C01791=1018.600,222.779,-127.632,168.817,51.228,159.725
C01792=1018.606,223.027,-127.658,168.821,51.221,159.724
C01793=1018.612,223.276,-127.684,168.825,51.214,159.724
C01794=1018.618,223.524,-127.710,168.829,51.207,159.723
C01795=1018.624,223.773,-127.736,168.833,51.201,159.722
C01796=1018.631,224.022,-127.763,168.836,51.194,159.721
C01797=1018.636,224.271,-127.789,168.841,51.188,159.721
C01798=1018.643,224.519,-127.815,168.846,51.181,159.720
C01799=1018.648,224.768,-127.841,168.849,51.174,159.719
C01800=1018.655,225.016,-127.867,168.854,51.168,159.719
C01801=1018.660,225.265,-127.893,168.857,51.161,159.718
C01802=1018.666,225.513,-127.919,168.862,51.155,159.717
C01803=1018.672,225.761,-127.945,168.865,51.148,159.716
C01804=1018.678,226.010,-127.971,168.870,51.141,159.716
C01805=1018.684,226.258,-127.997,168.873,51.135,159.715
C01806=1018.690,226.508,-128.024,168.877,51.128,159.714
C01807=1018.696,226.756,-128.050,168.881,51.122,159.714
C01808=1018.702,227.005,-128.077,168.886,51.115,159.713
C01809=1018.709,227.253,-128.103,168.889,51.109,159.712
C01810=1018.714,227.502,-128.129,168.894,51.102,159.712
C01811=1018.720,227.750,-128.156,168.897,51.096,159.711
C01812=1018.726,227.998,-128.182,168.902,51.090,159.710
C01813=1018.731,228.247,-128.209,168.906,51.083,159.710
C01814=1018.738,228.496,-128.236,168.910,51.077,159.709
C01815=1018.743,228.745,-128.262,168.914,51.071,159.709
C01816=1018.750,228.993,-128.288,168.918,51.064,159.708
C01817=1018.755,229.241,-128.314,168.922,51.058,159.707
C01818=1018.761,229.490,-128.341,168.927,51.051,159.706
C01819=1018.767,229.738,-128.368,168.930,51.045,159.706
C01820=1018.773,229.987,-128.395,168.935,51.039,159.705
C01821=1018.779,230.235,-128.421,168.939,51.033,159.705
C01822=1018.785,230.484,-128.448,168.942,51.026,159.704
C01823=1018.791,230.732,-128.475,168.947,51.020,159.703
C01824=1018.796,230.980,-128.501,168.951,51.014,159.703
C01825=1018.803,231.229,-128.528,168.955,51.007,159.702
C01826=1018.808,231.478,-128.554,168.959,51.001,159.701
C01827=1018.814,231.727,-128.581,168.964,50.995,159.701
C01828=1018.820,231.975,-128.608,168.967,50.989,159.700
C01829=1018.826,232.223,-128.635,168.971,50.983,159.699
C01830=1018.832,232.472,-128.662,168.976,50.976,159.699
C01831=1018.838,232.720,-128.689,168.979,50.970,159.698
C01832=1018.844,232.969,-128.715,168.984,50.964,159.698
C01833=1018.850,233.217,-128.742,168.988,50.958,159.697
C01834=1018.856,233.444,-128.766,168.992,50.952,159.697
C01835=1018.861,233.670,-128.790,168.996,50.947,159.696
C01836=1018.867,233.895,-128.815,169.000,50.941,159.695
C01837=1018.872,234.122,-128.839,169.003,50.936,159.695
C01838=1018.877,234.348,-128.864,169.007,50.930,159.694
C01839=1018.882,234.574,-128.888,169.011,50.924,159.694
C01840=1018.888,234.800,-128.913,169.015,50.919,159.693
C01841=1018.893,235.026,-128.937,169.019,50.913,159.693
C01842=1018.900,235.275,-128.964,169.022,50.907,159.692
C01843=1018.905,235.523,-128.991,169.027,50.901,159.692
C01844=1018.911,235.771,-129.018,169.031,50.895,159.691
C01845=1018.917,236.019,-129.045,169.034,50.889,159.690
C01846=1018.924,236.268,-129.072,169.040,50.883,159.690
C01847=1018.929,236.517,-129.098,169.043,50.877,159.689
C01848=1018.936,236.766,-129.125,169.047,50.871,159.688
C01849=1018.942,237.014,-129.153,169.052,50.864,159.688
C01850=1018.948,237.262,-129.179,169.056,50.859,159.687
C01851=1018.954,237.511,-129.206,169.060,50.852,159.687
C01852=1018.960,237.759,-129.234,169.064,50.846,159.686
C01853=1018.966,238.007,-129.260,169.068,50.840,159.686
C01854=1018.972,238.256,-129.287,169.073,50.834,159.685
C01855=1018.978,238.504,-129.314,169.077,50.828,159.684
C01856=1018.985,238.753,-129.342,169.080,50.822,159.684
C01857=1018.990,239.002,-129.369,169.085,50.817,159.683
C01858=1018.996,239.249,-129.396,169.089,50.810,159.683
C01859=1019.002,239.498,-129.423,169.093,50.805,159.682
C01860=1019.008,239.747,-129.450,169.098,50.799,159.682
C01861=1019.014,239.996,-129.478,169.102,50.793,159.681
C01862=1019.020,240.244,-129.505,169.106,50.787,159.681
C01863=1019.026,240.492,-129.532,169.111,50.781,159.680
C01864=1019.032,240.740,-129.561,169.114,50.775,159.680
C01865=1019.037,240.989,-129.587,169.119,50.770,159.679
C01866=1019.044,241.237,-129.615,169.123,50.764,159.678
C01867=1019.049,241.486,-129.642,169.127,50.758,159.678
C01868=1019.056,241.734,-129.670,169.131,50.752,159.677
C01869=1019.061,241.983,-129.697,169.135,50.747,159.677
C01870=1019.067,242.231,-129.725,169.140,50.741,159.676
C01871=1019.073,242.480,-129.752,169.144,50.735,159.676
C01872=1019.079,242.728,-129.780,169.148,50.730,159.675
C01873=1019.085,242.976,-129.807,169.153,50.723,159.675
C01874=1019.091,243.225,-129.834,169.157,50.718,159.674
C01875=1019.097,243.473,-129.862,169.161,50.712,159.674
C01876=1019.102,243.721,-129.890,169.165,50.707,159.673
C01877=1019.109,243.970,-129.918,169.170,50.701,159.673
C01878=1019.114,244.218,-129.946,169.174,50.695,159.672
C01879=1019.121,244.467,-129.973,169.178,50.690,159.672
C01880=1019.126,244.715,-130.001,169.182,50.684,159.671
C01881=1019.132,244.964,-130.029,169.187,50.679,159.671
C01882=1019.138,245.211,-130.057,169.191,50.673,159.670
C01883=1019.144,245.460,-130.085,169.195,50.667,159.670
C01884=1019.149,245.708,-130.113,169.199,50.662,159.669
C01885=1019.156,245.957,-130.140,169.203,50.657,159.669
C01886=1019.161,246.205,-130.168,169.208,50.651,159.669
C01887=1019.168,246.454,-130.196,169.213,50.645,159.668
C01888=1019.174,246.703,-130.224,169.217,50.640,159.668
C01889=1019.179,246.951,-130.252,169.221,50.635,159.667
C01890=1019.186,247.199,-130.280,169.226,50.628,159.667
C01891=1019.191,247.447,-130.308,169.230,50.623,159.666
C01892=1019.197,247.696,-130.336,169.234,50.618,159.666
C01893=1019.203,247.944,-130.363,169.238,50.612,159.665
C01894=1019.208,248.167,-130.389,169.242,50.608,159.665
C01895=1019.213,248.390,-130.413,169.245,50.602,159.664
C01896=1019.219,248.612,-130.438,169.250,50.598,159.664
C01897=1019.224,248.835,-130.464,169.253,50.593,159.663
C01898=1019.230,249.058,-130.489,169.258,50.588,159.663
C01899=1019.235,249.280,-130.514,169.262,50.583,159.663
C01900=1019.241,249.504,-130.539,169.265,50.578,159.662
C01901=1019.246,249.726,-130.564,169.269,50.573,159.662
C01902=1019.252,249.975,-130.592,169.273,50.568,159.661
C01903=1019.258,250.224,-130.620,169.278,50.562,159.661
C01904=1019.264,250.472,-130.648,169.282,50.557,159.660
C01905=1019.271,250.720,-130.677,169.287,50.551,159.660
C01906=1019.276,250.968,-130.705,169.291,50.546,159.660
C01907=1019.282,251.216,-130.733,169.295,50.541,159.659
C01908=1019.288,251.465,-130.761,169.300,50.536,159.659
C01909=1019.294,251.714,-130.789,169.305,50.530,159.659
C01910=1019.300,251.962,-130.817,169.309,50.525,159.658
C01911=1019.306,252.210,-130.845,169.313,50.519,159.658
C01912=1019.312,252.459,-130.873,169.317,50.514,159.657
C01913=1019.319,252.707,-130.902,169.321,50.509,159.657
C01914=1019.325,252.955,-130.930,169.326,50.503,159.656
C01915=1019.331,253.203,-130.958,169.331,50.498,159.656
C01916=1019.337,253.452,-130.986,169.335,50.493,159.656
C01917=1019.344,253.700,-131.014,169.339,50.488,159.655
C01918=1019.350,253.949,-131.043,169.343,50.482,159.655
C01919=1019.356,254.196,-131.070,169.348,50.477,159.654
C01920=1019.362,254.445,-131.098,169.352,50.471,159.654
C01921=1019.368,254.693,-131.128,169.357,50.466,159.653
C01922=1019.375,254.942,-131.155,169.361,50.461,159.653
C01923=1019.380,255.191,-131.184,169.366,50.455,159.653
C01924=1019.386,255.439,-131.212,169.370,50.450,159.652
C01925=1019.393,255.686,-131.240,169.375,50.445,159.652
C01926=1019.399,255.935,-131.268,169.379,50.440,159.651
C01927=1019.405,256.184,-131.297,169.383,50.435,159.651
C01928=1019.412,256.432,-131.325,169.388,50.429,159.650
C01929=1019.418,256.680,-131.353,169.393,50.424,159.650
C01930=1019.423,256.929,-131.381,169.397,50.419,159.650
C01931=1019.430,257.176,-131.410,169.401,50.414,159.649
C01932=1019.436,257.425,-131.438,169.406,50.409,159.649
C01933=1019.442,257.673,-131.467,169.411,50.403,159.649
C01934=1019.449,257.922,-131.495,169.415,50.398,159.648
C01935=1019.455,258.170,-131.524,169.419,50.393,159.648
C01936=1019.461,258.419,-131.552,169.423,50.388,159.647
C01937=1019.468,258.667,-131.580,169.429,50.383,159.647
C01938=1019.474,258.915,-131.609,169.433,50.378,159.647
C01939=1019.480,259.164,-131.637,169.437,50.372,159.646
C01940=1019.487,259.412,-131.666,169.442,50.368,159.646
C01941=1019.492,259.660,-131.694,169.446,50.362,159.645
C01942=1019.498,259.908,-131.723,169.451,50.357,159.645
C01943=1019.505,260.156,-131.752,169.456,50.352,159.645
C01944=1019.511,260.405,-131.780,169.460,50.347,159.645
C01945=1019.517,260.653,-131.809,169.464,50.342,159.644
C01946=1019.523,260.901,-131.838,169.469,50.337,159.644
C01947=1019.529,261.149,-131.867,169.473,50.333,159.644
C01948=1019.535,261.398,-131.896,169.477,50.327,159.643
C01949=1019.542,261.646,-131.925,169.482,50.323,159.643
C01950=1019.548,261.894,-131.954,169.487,50.318,159.643
C01951=1019.554,262.142,-131.983,169.492,50.313,159.642
C01952=1019.560,262.390,-132.012,169.496,50.308,159.642
C01953=1019.566,262.639,-132.040,169.501,50.303,159.642
C01954=1019.571,262.861,-132.066,169.504,50.299,159.641
C01955=1019.577,263.083,-132.092,169.509,50.294,159.641
C01956=1019.582,263.305,-132.118,169.513,50.290,159.641
C01957=1019.588,263.527,-132.144,169.517,50.286,159.641
C01958=1019.593,263.749,-132.170,169.521,50.281,159.640
C01959=1019.599,263.970,-132.196,169.525,50.277,159.640
C01960=1019.605,264.192,-132.222,169.529,50.272,159.639
C01961=1019.610,264.415,-132.248,169.534,50.268,159.639
C01962=1019.616,264.663,-132.277,169.538,50.263,159.639
C01963=1019.622,264.911,-132.306,169.542,50.259,159.639
C01964=1019.629,265.159,-132.335,169.547,50.254,159.638
C01965=1019.635,265.407,-132.364,169.551,50.249,159.638
C01966=1019.640,265.656,-132.394,169.556,50.245,159.638
C01967=1019.647,265.904,-132.423,169.560,50.240,159.638
C01968=1019.653,266.152,-132.452,169.566,50.235,159.637
C01969=1019.659,266.400,-132.481,169.570,50.230,159.637
C01970=1019.665,266.648,-132.510,169.575,50.226,159.637
C01971=1019.671,266.896,-132.540,169.579,50.221,159.637
C01972=1019.678,267.145,-132.570,169.584,50.216,159.636
C01973=1019.684,267.393,-132.599,169.589,50.212,159.636
C01974=1019.691,267.641,-132.628,169.593,50.207,159.636
C01975=1019.696,267.890,-132.657,169.598,50.202,159.635
C01976=1019.702,268.138,-132.686,169.602,50.198,159.635
C01977=1019.709,268.385,-132.716,169.607,50.193,159.635
C01978=1019.714,268.634,-132.746,169.612,50.188,159.635
C01979=1019.721,268.882,-132.775,169.617,50.183,159.634
C01980=1019.727,269.131,-132.804,169.621,50.179,159.634
C01981=1019.734,269.379,-132.833,169.626,50.174,159.634
C01982=1019.740,269.627,-132.864,169.630,50.170,159.634
C01983=1019.746,269.875,-132.893,169.635,50.165,159.633
C01984=1019.751,270.123,-132.922,169.639,50.160,159.633
C01985=1019.758,270.371,-132.952,169.644,50.156,159.633
C01986=1019.765,270.619,-132.981,169.649,50.152,159.633
C01987=1019.770,270.867,-133.012,169.653,50.147,159.632
C01988=1019.777,271.115,-133.041,169.658,50.142,159.632
C01989=1019.782,271.364,-133.070,169.662,50.138,159.632
C01990=1019.789,271.611,-133.100,169.668,50.133,159.632
C01991=1019.796,271.860,-133.130,169.673,50.129,159.632
C01992=1019.801,272.108,-133.160,169.677,50.124,159.631
C01993=1019.808,272.356,-133.189,169.682,50.120,159.631
C01994=1019.814,272.604,-133.219,169.687,50.116,159.631
C01995=1019.820,272.853,-133.249,169.691,50.111,159.631
C01996=1019.826,273.101,-133.279,169.696,50.106,159.630
C01997=1019.832,273.349,-133.308,169.701,50.102,159.630
C01998=1019.838,273.597,-133.339,169.705,50.098,159.630
C01999=1019.845,273.845,-133.368,169.710,50.093,159.630
C02000=1019.851,274.093,-133.398,169.715,50.089,159.630
C02001=1019.857,274.341,-133.428,169.719,50.085,159.629
C02002=1019.864,274.590,-133.458,169.724,50.081,159.629
C02003=1019.870,274.837,-133.488,169.729,50.076,159.629
C02004=1019.876,275.086,-133.517,169.733,50.071,159.629
C02005=1019.882,275.333,-133.547,169.739,50.067,159.629
C02006=1019.889,275.582,-133.578,169.744,50.062,159.628
C02007=1019.895,275.830,-133.607,169.749,50.058,159.628
C02008=1019.901,276.078,-133.637,169.753,50.054,159.628
C02009=1019.907,276.326,-133.668,169.758,50.050,159.628
C02010=1019.914,276.574,-133.698,169.763,50.045,159.628
C02011=1019.920,276.823,-133.728,169.768,50.041,159.628
C02012=1019.926,277.071,-133.758,169.772,50.037,159.627
C02013=1019.932,277.318,-133.788,169.777,50.033,159.627
C02014=1019.938,277.542,-133.816,169.781,50.029,159.627
C02015=1019.943,277.767,-133.843,169.786,50.025,159.627
C02016=1019.949,277.991,-133.870,169.790,50.021,159.627
C02017=1019.955,278.215,-133.898,169.795,50.017,159.627
C02018=1019.960,278.440,-133.925,169.799,50.014,159.627
C02019=1019.966,278.664,-133.953,169.804,50.010,159.626
C02020=1019.971,278.888,-133.980,169.808,50.006,159.626
C02021=1019.977,279.112,-134.007,169.813,50.002,159.626
C02022=1019.983,279.361,-134.038,169.817,49.998,159.626
C02023=1019.990,279.608,-134.068,169.822,49.994,159.626
C02024=1019.996,279.857,-134.099,169.827,49.990,159.626
C02025=1020.002,280.105,-134.129,169.832,49.986,159.626
C02026=1020.008,280.353,-134.160,169.837,49.982,159.626
C02027=1020.014,280.601,-134.190,169.841,49.977,159.625
C02028=1020.021,280.849,-134.220,169.846,49.973,159.625
C02029=1020.027,281.097,-134.250,169.851,49.969,159.625
C02030=1020.033,281.345,-134.281,169.856,49.965,159.625
C02031=1020.039,281.593,-134.311,169.861,49.961,159.625
C02032=1020.046,281.841,-134.341,169.866,49.957,159.625
C02033=1020.053,282.089,-134.373,169.870,49.953,159.625
C02034=1020.058,282.337,-134.403,169.875,49.949,159.624
C02035=1020.065,282.585,-134.434,169.880,49.945,159.624
C02036=1020.071,282.834,-134.464,169.885,49.941,159.624
C02037=1020.078,283.081,-134.494,169.890,49.937,159.624
C02038=1020.084,283.330,-134.525,169.895,49.933,159.624
C02039=1020.090,283.577,-134.556,169.900,49.929,159.624
C02040=1020.097,283.825,-134.587,169.906,49.924,159.624
C02041=1020.103,284.073,-134.616,169.910,49.920,159.624
C02042=1020.110,284.321,-134.647,169.915,49.916,159.624
C02043=1020.117,284.569,-134.679,169.920,49.912,159.624
C02044=1020.122,284.817,-134.709,169.925,49.909,159.623
C02045=1020.129,285.066,-134.740,169.930,49.905,159.623
C02046=1020.135,285.313,-134.771,169.935,49.901,159.623
C02047=1020.141,285.561,-134.801,169.940,49.897,159.623
C02048=1020.147,285.809,-134.833,169.945,49.893,159.623
C02049=1020.154,286.057,-134.863,169.950,49.889,159.623
C02050=1020.161,286.305,-134.895,169.955,49.886,159.623
C02051=1020.166,286.553,-134.925,169.960,49.882,159.623
C02052=1020.173,286.801,-134.956,169.965,49.878,159.623
C02053=1020.180,287.049,-134.987,169.970,49.874,159.623
C02054=1020.186,287.296,-135.018,169.975,49.870,159.623
C02055=1020.192,287.545,-135.049,169.980,49.866,159.623
C02056=1020.199,287.793,-135.080,169.985,49.863,159.623
C02057=1020.205,288.041,-135.111,169.990,49.859,159.623
C02058=1020.211,288.289,-135.142,169.995,49.855,159.623
C02059=1020.218,288.537,-135.173,170.000,49.851,159.623
C02060=1020.224,288.784,-135.204,170.005,49.847,159.623
C02061=1020.231,289.032,-135.235,170.010,49.844,159.623
C02062=1020.237,289.281,-135.266,170.015,49.840,159.622
C02063=1020.244,289.529,-135.298,170.020,49.836,159.623
C02064=1020.250,289.776,-135.329,170.025,49.832,159.622
C02065=1020.256,290.025,-135.360,170.031,49.828,159.622
C02066=1020.262,290.273,-135.391,170.036,49.824,159.622
C02067=1020.269,290.521,-135.423,170.041,49.821,159.622
C02068=1020.275,290.768,-135.454,170.046,49.817,159.622
C02069=1020.282,291.016,-135.485,170.052,49.814,159.622
C02070=1020.288,291.264,-135.516,170.057,49.810,159.622
C02071=1020.295,291.512,-135.547,170.061,49.806,159.622
C02072=1020.302,291.760,-135.579,170.067,49.803,159.622
C02073=1020.307,292.007,-135.611,170.072,49.799,159.622
C02074=1020.314,292.238,-135.639,170.076,49.796,159.622
C02075=1020.320,292.469,-135.669,170.081,49.792,159.622
C02076=1020.325,292.699,-135.698,170.086,49.788,159.622
C02077=1020.332,292.929,-135.727,170.091,49.786,159.622
C02078=1020.338,293.160,-135.757,170.096,49.782,159.622
C02079=1020.343,293.390,-135.786,170.101,49.778,159.622
C02080=1020.349,293.620,-135.815,170.105,49.775,159.622
C02081=1020.355,293.851,-135.845,170.110,49.772,159.623
C02082=1020.361,294.098,-135.877,170.116,49.769,159.623
C02083=1020.367,294.346,-135.908,170.121,49.765,159.623
C02084=1020.373,294.595,-135.940,170.126,49.762,159.623
C02085=1020.380,294.842,-135.972,170.131,49.758,159.623
C02086=1020.386,295.090,-136.004,170.136,49.755,159.623
C02087=1020.392,295.338,-136.037,170.141,49.751,159.623
C02088=1020.399,295.585,-136.068,170.147,49.748,159.623
C02089=1020.405,295.834,-136.100,170.152,49.745,159.623
C02090=1020.412,296.081,-136.132,170.157,49.741,159.623
C02091=1020.418,296.329,-136.164,170.163,49.738,159.623
C02092=1020.424,296.577,-136.195,170.168,49.734,159.623
C02093=1020.431,296.825,-136.228,170.173,49.731,159.623
C02094=1020.437,297.073,-136.260,170.178,49.728,159.623
C02095=1020.443,297.321,-136.291,170.183,49.724,159.623
C02096=1020.450,297.568,-136.324,170.189,49.721,159.623
C02097=1020.456,297.816,-136.356,170.194,49.718,159.624
C02098=1020.462,298.064,-136.388,170.199,49.714,159.623
C02099=1020.469,298.312,-136.420,170.204,49.711,159.624
C02100=1020.475,298.560,-136.452,170.210,49.707,159.624
C02101=1020.482,298.808,-136.485,170.215,49.704,159.624
C02102=1020.488,299.055,-136.516,170.220,49.701,159.624
C02103=1020.495,299.303,-136.549,170.226,49.698,159.624
C02104=1020.501,299.551,-136.580,170.231,49.694,159.624
C02105=1020.507,299.799,-136.612,170.236,49.691,159.624
C02106=1020.514,300.047,-136.645,170.241,49.688,159.624
C02107=1020.521,300.294,-136.677,170.247,49.685,159.624
C02108=1020.527,300.542,-136.709,170.252,49.681,159.624
C02109=1020.534,300.790,-136.741,170.257,49.678,159.625
C02110=1020.540,301.038,-136.773,170.263,49.675,159.625
C02111=1020.547,301.285,-136.805,170.268,49.671,159.625
C02112=1020.553,301.533,-136.837,170.273,49.668,159.625
C02113=1020.559,301.781,-136.870,170.279,49.665,159.625
C02114=1020.567,302.029,-136.903,170.284,49.662,159.625
C02115=1020.573,302.277,-136.935,170.289,49.658,159.625
C02116=1020.580,302.524,-136.967,170.295,49.656,159.625
C02117=1020.586,302.772,-137.000,170.300,49.653,159.626
C02118=1020.592,303.020,-137.032,170.305,49.649,159.626
C02119=1020.599,303.267,-137.064,170.311,49.646,159.626
C02120=1020.606,303.516,-137.097,170.317,49.642,159.626
C02121=1020.613,303.763,-137.129,170.322,49.639,159.626
C02122=1020.619,304.011,-137.161,170.328,49.637,159.626
C02123=1020.625,304.259,-137.194,170.333,49.633,159.626
C02124=1020.632,304.506,-137.226,170.339,49.630,159.627
C02125=1020.639,304.754,-137.259,170.344,49.627,159.627
C02126=1020.646,305.002,-137.291,170.349,49.624,159.627
C02127=1020.652,305.250,-137.323,170.355,49.621,159.627
C02128=1020.658,305.497,-137.356,170.360,49.618,159.627
C02129=1020.666,305.745,-137.389,170.365,49.614,159.627
C02130=1020.672,305.993,-137.421,170.371,49.612,159.628
C02131=1020.679,306.240,-137.453,170.377,49.608,159.628
C02132=1020.686,306.489,-137.487,170.383,49.605,159.628
C02133=1020.693,306.736,-137.519,170.388,49.602,159.628
C02134=1020.699,306.976,-137.550,170.394,49.599,159.628
C02135=1020.706,307.214,-137.582,170.399,49.596,159.628
C02136=1020.712,307.454,-137.613,170.404,49.594,159.628
C02137=1020.719,307.693,-137.645,170.409,49.590,159.629
C02138=1020.725,307.932,-137.676,170.415,49.588,159.629
C02139=1020.732,308.171,-137.708,170.420,49.584,159.629
C02140=1020.739,308.410,-137.739,170.426,49.582,159.629
C02141=1020.745,308.650,-137.771,170.431,49.579,159.629
C02142=1020.752,308.897,-137.804,170.437,49.576,159.630
C02143=1020.759,309.144,-137.836,170.442,49.573,159.630
C02144=1020.766,309.393,-137.869,170.447,49.569,159.630
C02145=1020.773,309.640,-137.902,170.454,49.567,159.630
C02146=1020.780,309.888,-137.935,170.459,49.563,159.630
C02147=1020.786,310.135,-137.968,170.465,49.561,159.631
C02148=1020.792,310.383,-138.001,170.470,49.558,159.631
C02149=1020.800,310.631,-138.035,170.476,49.555,159.631
C02150=1020.806,310.878,-138.067,170.481,49.552,159.631
C02151=1020.812,311.125,-138.101,170.487,49.550,159.632
C02152=1020.819,311.374,-138.135,170.493,49.547,159.632
C02153=1020.825,311.621,-138.168,170.498,49.544,159.632
C02154=1020.832,311.869,-138.201,170.504,49.542,159.632
C02155=1020.838,312.116,-138.235,170.509,49.539,159.633
C02156=1020.845,312.365,-138.268,170.515,49.536,159.633
C02157=1020.852,312.612,-138.302,170.521,49.533,159.633
C02158=1020.858,312.859,-138.335,170.526,49.531,159.633
C02159=1020.865,313.107,-138.368,170.532,49.528,159.634
C02160=1020.871,313.354,-138.402,170.538,49.526,159.634
C02161=1020.878,313.602,-138.435,170.544,49.523,159.634
C02162=1020.884,313.849,-138.469,170.550,49.520,159.635
C02163=1020.892,314.097,-138.503,170.556,49.517,159.635
C02164=1020.898,314.345,-138.537,170.561,49.515,159.635
C02165=1020.904,314.593,-138.570,170.567,49.512,159.636
C02166=1020.912,314.840,-138.604,170.573,49.510,159.636
C02167=1020.918,315.087,-138.637,170.578,49.507,159.636
C02168=1020.924,315.336,-138.671,170.584,49.504,159.636
C02169=1020.931,315.583,-138.704,170.590,49.502,159.637
C02170=1020.938,315.831,-138.738,170.595,49.499,159.637
C02171=1020.945,316.078,-138.772,170.601,49.497,159.637
C02172=1020.951,316.325,-138.806,170.608,49.494,159.638
C02173=1020.958,316.573,-138.840,170.613,49.491,159.638
C02174=1020.965,316.821,-138.873,170.619,49.488,159.638
C02175=1020.971,317.069,-138.907,170.625,49.486,159.639
C02176=1020.978,317.316,-138.941,170.630,49.483,159.639
C02177=1020.986,317.564,-138.975,170.636,49.481,159.639
C02178=1020.992,317.811,-139.008,170.642,49.478,159.639
C02179=1020.999,318.059,-139.043,170.649,49.476,159.640
C02180=1021.006,318.307,-139.076,170.655,49.473,159.640
C02181=1021.013,318.554,-139.110,170.660,49.471,159.641
C02182=1021.020,318.801,-139.144,170.666,49.468,159.641
C02183=1021.026,319.049,-139.178,170.672,49.465,159.641
C02184=1021.033,319.297,-139.212,170.678,49.463,159.642
C02185=1021.040,319.545,-139.246,170.683,49.461,159.642
C02186=1021.046,319.792,-139.280,170.690,49.458,159.642
C02187=1021.054,320.040,-139.314,170.696,49.456,159.643
C02188=1021.061,320.287,-139.347,170.702,49.453,159.643
C02189=1021.068,320.534,-139.382,170.707,49.451,159.643
C02190=1021.075,320.782,-139.416,170.713,49.448,159.644
C02191=1021.082,321.030,-139.450,170.719,49.446,159.644
C02192=1021.088,321.277,-139.484,170.726,49.443,159.644
C02193=1021.096,321.525,-139.518,170.732,49.441,159.645
C02194=1021.102,321.767,-139.551,170.737,49.439,159.645
C02195=1021.109,322.008,-139.585,170.743,49.436,159.645
C02196=1021.116,322.250,-139.618,170.749,49.434,159.646
C02197=1021.123,322.492,-139.651,170.755,49.432,159.646
C02198=1021.130,322.733,-139.685,170.761,49.430,159.647
C02199=1021.137,322.975,-139.718,170.766,49.427,159.647
C02200=1021.144,323.217,-139.751,170.772,49.425,159.647
C02201=1021.151,323.458,-139.785,170.778,49.423,159.648
C02202=1021.158,323.706,-139.819,170.785,49.420,159.648
C02203=1021.164,323.954,-139.853,170.791,49.418,159.649
C02204=1021.172,324.201,-139.888,170.797,49.416,159.649
C02205=1021.179,324.448,-139.922,170.802,49.413,159.649
C02206=1021.186,324.696,-139.957,170.809,49.411,159.650
C02207=1021.193,324.944,-139.991,170.815,49.408,159.650
C02208=1021.201,325.192,-140.025,170.821,49.406,159.651
C02209=1021.207,325.439,-140.060,170.827,49.404,159.651
C02210=1021.215,325.687,-140.094,170.834,49.401,159.652
C02211=1021.222,325.934,-140.128,170.840,49.399,159.652
C02212=1021.229,326.182,-140.162,170.846,49.397,159.652
C02213=1021.236,326.429,-140.197,170.852,49.395,159.653
C02214=1021.244,326.676,-140.232,170.859,49.393,159.653
C02215=1021.250,326.924,-140.266,170.865,49.391,159.654
C02216=1021.258,327.171,-140.301,170.870,49.388,159.654
C02217=1021.264,327.418,-140.336,170.876,49.386,159.655
C02218=1021.272,327.667,-140.371,170.882,49.384,159.655
C02219=1021.278,327.914,-140.406,170.889,49.382,159.656
C02220=1021.286,328.162,-140.440,170.895,49.380,159.656
C02221=1021.292,328.409,-140.475,170.902,49.378,159.657
C02222=1021.299,328.656,-140.511,170.908,49.376,159.657
C02223=1021.306,328.904,-140.546,170.915,49.374,159.658
C02224=1021.313,329.151,-140.580,170.921,49.372,159.658
C02225=1021.321,329.399,-140.616,170.927,49.370,159.659
C02226=1021.328,329.646,-140.651,170.933,49.368,159.659
C02227=1021.334,329.894,-140.686,170.940,49.366,159.660
C02228=1021.342,330.141,-140.720,170.946,49.364,159.660
C02229=1021.349,330.388,-140.756,170.952,49.362,159.661
C02230=1021.356,330.636,-140.791,170.958,49.360,159.661
C02231=1021.363,330.883,-140.826,170.965,49.357,159.662
C02232=1021.370,331.130,-140.861,170.971,49.355,159.662
C02233=1021.378,331.378,-140.896,170.977,49.354,159.663
C02234=1021.384,331.626,-140.931,170.983,49.352,159.663
C02235=1021.392,331.873,-140.967,170.990,49.350,159.664
C02236=1021.399,332.120,-141.002,170.996,49.348,159.664
C02237=1021.406,332.368,-141.037,171.002,49.346,159.665
C02238=1021.413,332.615,-141.072,171.009,49.344,159.665
C02239=1021.421,332.863,-141.108,171.015,49.342,159.666
C02240=1021.428,333.110,-141.143,171.022,49.340,159.666
C02241=1021.435,333.357,-141.178,171.028,49.339,159.667
C02242=1021.442,333.605,-141.214,171.035,49.336,159.668
C02243=1021.450,333.852,-141.250,171.041,49.335,159.668
C02244=1021.456,334.099,-141.285,171.047,49.333,159.669
C02245=1021.464,334.347,-141.321,171.054,49.331,159.669
C02246=1021.471,334.594,-141.356,171.061,49.329,159.670
C02247=1021.478,334.841,-141.392,171.067,49.327,159.670
C02248=1021.485,335.089,-141.428,171.074,49.326,159.671
C02249=1021.492,335.335,-141.463,171.080,49.324,159.672
C02250=1021.500,335.584,-141.499,171.087,49.322,159.672
C02251=1021.507,335.830,-141.535,171.094,49.320,159.673
C02252=1021.514,336.078,-141.570,171.100,49.319,159.674
C02253=1021.521,336.325,-141.606,171.106,49.317,159.674
C02254=1021.528,336.565,-141.642,171.112,49.316,159.675
C02255=1021.535,336.805,-141.676,171.118,49.314,159.675
C02256=1021.542,337.044,-141.711,171.126,49.312,159.676
C02257=1021.549,337.283,-141.746,171.132,49.310,159.676
C02258=1021.556,337.523,-141.780,171.138,49.309,159.677
C02259=1021.563,337.763,-141.815,171.144,49.307,159.678
C02260=1021.570,338.002,-141.849,171.151,49.305,159.678
C02261=1021.578,338.242,-141.885,171.157,49.304,159.679
C02262=1021.585,338.488,-141.920,171.164,49.302,159.679
C02263=1021.592,338.736,-141.956,171.170,49.301,159.680
C02264=1021.599,338.983,-141.992,171.178,49.299,159.681
C02265=1021.607,339.231,-142.028,171.184,49.297,159.681
C02266=1021.615,339.478,-142.064,171.190,49.296,159.682
C02267=1021.622,339.725,-142.100,171.198,49.294,159.683
C02268=1021.629,339.972,-142.136,171.204,49.293,159.683
C02269=1021.636,340.220,-142.173,171.210,49.291,159.684
C02270=1021.643,340.467,-142.209,171.218,49.290,159.685
C02271=1021.651,340.714,-142.245,171.224,49.288,159.685
C02272=1021.659,340.962,-142.281,171.231,49.286,159.686
C02273=1021.665,341.209,-142.318,171.238,49.285,159.687
C02274=1021.673,341.456,-142.354,171.244,49.283,159.687
C02275=1021.680,341.704,-142.390,171.251,49.282,159.688
C02276=1021.688,341.950,-142.427,171.258,49.280,159.689
C02277=1021.695,342.197,-142.464,171.265,49.279,159.690
C02278=1021.702,342.445,-142.500,171.271,49.277,159.690
C02279=1021.710,342.692,-142.536,171.279,49.276,159.691
C02280=1021.717,342.940,-142.573,171.285,49.274,159.692
C02281=1021.724,343.186,-142.609,171.292,49.273,159.692
C02282=1021.732,343.434,-142.646,171.299,49.271,159.693
C02283=1021.739,343.681,-142.682,171.306,49.271,159.694
C02284=1021.747,343.928,-142.719,171.313,49.269,159.695
C02285=1021.755,344.176,-142.756,171.320,49.268,159.695
C02286=1021.762,344.423,-142.793,171.327,49.266,159.696
C02287=1021.769,344.670,-142.829,171.333,49.265,159.697
C02288=1021.777,344.917,-142.865,171.341,49.263,159.698
C02289=1021.784,345.164,-142.903,171.347,49.262,159.698
C02290=1021.792,345.412,-142.939,171.354,49.261,159.699
C02291=1021.799,345.659,-142.976,171.361,49.259,159.700
C02292=1021.806,345.906,-143.013,171.368,49.258,159.701
C02293=1021.814,346.153,-143.050,171.375,49.257,159.701
C02294=1021.822,346.400,-143.087,171.382,49.256,159.702
C02295=1021.829,346.648,-143.123,171.389,49.254,159.703
C02296=1021.837,346.894,-143.160,171.396,49.253,159.704
C02297=1021.844,347.142,-143.197,171.403,49.252,159.705
C02298=1021.852,347.389,-143.234,171.411,49.251,159.705
C02299=1021.859,347.636,-143.272,171.417,49.249,159.706
C02300=1021.867,347.883,-143.308,171.425,49.248,159.707
C02301=1021.874,348.131,-143.345,171.431,49.247,159.708
C02302=1021.882,348.378,-143.382,171.439,49.245,159.708
C02303=1021.890,348.625,-143.420,171.446,49.245,159.709
C02304=1021.898,348.871,-143.457,171.453,49.244,159.710
C02305=1021.905,349.119,-143.494,171.460,49.242,159.711
C02306=1021.912,349.366,-143.532,171.467,49.241,159.712
C02307=1021.920,349.613,-143.569,171.474,49.240,159.713
C02308=1021.927,349.860,-143.606,171.482,49.239,159.714
C02309=1021.935,350.108,-143.644,171.488,49.238,159.714
C02310=1021.943,350.354,-143.681,171.496,49.237,159.715
C02311=1021.950,350.601,-143.719,171.503,49.236,159.716
C02312=1021.958,350.848,-143.755,171.510,49.235,159.717
C02313=1021.966,351.095,-143.793,171.518,49.234,159.718
C02314=1021.973,351.333,-143.829,171.524,49.232,159.719
C02315=1021.981,351.571,-143.865,171.531,49.232,159.719
C02316=1021.988,351.809,-143.902,171.539,49.231,159.720
C02317=1021.995,352.047,-143.938,171.546,49.230,159.721
C02318=1022.003,352.286,-143.974,171.552,49.229,159.722
C02319=1022.010,352.524,-144.010,171.560,49.228,159.723
C02320=1022.018,352.761,-144.046,171.566,49.227,159.724
C02321=1022.026,352.999,-144.083,171.574,49.226,159.725
C02322=1022.033,353.246,-144.120,171.581,49.225,159.726
C02323=1022.040,353.493,-144.158,171.589,49.224,159.727
C02324=1022.049,353.740,-144.196,171.596,49.222,159.727
C02325=1022.056,353.987,-144.233,171.603,49.222,159.728
C02326=1022.064,354.234,-144.271,171.610,49.221,159.729
C02327=1022.072,354.481,-144.309,171.619,49.220,159.730
C02328=1022.080,354.728,-144.347,171.625,49.220,159.731
C02329=1022.088,354.976,-144.385,171.633,49.219,159.732
C02330=1022.095,355.222,-144.423,171.641,49.218,159.733
C02331=1022.103,355.469,-144.461,171.648,49.217,159.734
C02332=1022.111,355.716,-144.499,171.655,49.216,159.735
C02333=1022.119,355.963,-144.537,171.663,49.215,159.736
C02334=1022.127,356.210,-144.575,171.670,49.215,159.737
C02335=1022.134,356.457,-144.613,171.678,49.214,159.738
C02336=1022.142,356.704,-144.651,171.686,49.213,159.739
C02337=1022.150,356.951,-144.690,171.692,49.212,159.740
C02338=1022.158,357.198,-144.727,171.700,49.211,159.741
C02339=1022.166,357.445,-144.765,171.708,49.210,159.742
C02340=1022.174,357.692,-144.804,171.716,49.209,159.743
C02341=1022.182,357.939,-144.842,171.723,49.209,159.744
C02342=1022.190,358.186,-144.881,171.731,49.208,159.745
C02343=1022.198,358.432,-144.919,171.739,49.207,159.746
C02344=1022.206,358.680,-144.958,171.747,49.207,159.747
C02345=1022.213,358.926,-144.996,171.753,49.206,159.748
C02346=1022.221,359.173,-145.035,171.761,49.206,159.749
C02347=1022.230,359.420,-145.072,171.769,49.205,159.750
C02348=1022.238,359.667,-145.111,171.777,49.204,159.751
C02349=1022.246,359.914,-145.149,171.785,49.203,159.752
C02350=1022.254,360.161,-145.188,171.792,49.203,159.753
C02351=1022.261,360.408,-145.227,171.800,49.202,159.754
C02352=1022.269,360.655,-145.265,171.808,49.201,159.755
C02353=1022.277,360.901,-145.304,171.816,49.201,159.756
C02354=1022.285,361.148,-145.343,171.823,49.200,159.757
C02355=1022.293,361.396,-145.382,171.831,49.200,159.758
C02356=1022.301,361.642,-145.421,171.839,49.199,159.759
C02357=1022.309,361.889,-145.460,171.847,49.199,159.760
C02358=1022.317,362.136,-145.498,171.855,49.199,159.762
C02359=1022.325,362.382,-145.537,171.863,49.198,159.762
C02360=1022.333,362.629,-145.576,171.870,49.197,159.764
C02361=1022.341,362.876,-145.615,171.878,49.197,159.765
C02362=1022.349,363.123,-145.654,171.886,49.197,159.766
C02363=1022.357,363.370,-145.694,171.894,49.196,159.767
C02364=1022.365,363.617,-145.732,171.902,49.196,159.768
C02365=1022.373,363.863,-145.771,171.911,49.195,159.769
C02366=1022.381,364.110,-145.810,171.919,49.195,159.770
C02367=1022.390,364.357,-145.849,171.926,49.195,159.771
C02368=1022.398,364.604,-145.889,171.934,49.194,159.773
C02369=1022.406,364.851,-145.928,171.942,49.194,159.774
C02370=1022.414,365.098,-145.967,171.950,49.193,159.775
C02371=1022.422,365.344,-146.006,171.958,49.193,159.776
C02372=1022.431,365.592,-146.045,171.966,49.192,159.777
C02373=1022.438,365.837,-146.084,171.974,49.192,159.778
C02374=1022.447,366.079,-146.123,171.982,49.192,159.779
C02375=1022.455,366.321,-146.161,171.991,49.191,159.781
C02376=1022.463,366.562,-146.200,171.999,49.191,159.782
C02377=1022.471,366.804,-146.238,172.006,49.191,159.783
C02378=1022.479,367.044,-146.277,172.014,49.190,159.784
C02379=1022.487,367.286,-146.315,172.022,49.190,159.785
C02380=1022.495,367.528,-146.354,172.030,49.190,159.786
C02381=1022.504,367.769,-146.393,172.039,49.189,159.788
C02382=1022.512,368.015,-146.432,172.047,49.189,159.789
C02383=1022.520,368.262,-146.472,172.055,49.189,159.790
C02384=1022.529,368.509,-146.511,172.063,49.189,159.791
C02385=1022.536,368.756,-146.551,172.072,49.189,159.793
C02386=1022.545,369.002,-146.590,172.080,49.188,159.794
C02387=1022.553,369.249,-146.631,172.088,49.188,159.795
C02388=1022.562,369.496,-146.671,172.096,49.188,159.796
C02389=1022.569,369.743,-146.711,172.105,49.188,159.798
C02390=1022.578,369.989,-146.751,172.113,49.188,159.799
C02391=1022.586,370.236,-146.791,172.121,49.188,159.800
C02392=1022.594,370.482,-146.830,172.130,49.188,159.801
C02393=1022.602,370.729,-146.871,172.138,49.188,159.803
C02394=1022.612,370.976,-146.910,172.146,49.188,159.804
C02395=1022.620,371.222,-146.951,172.155,49.188,159.805
C02396=1022.628,371.469,-146.990,172.164,49.187,159.806
C02397=1022.636,371.715,-147.031,172.172,49.187,159.808
C02398=1022.645,371.962,-147.071,172.181,49.187,159.809
C02399=1022.653,372.209,-147.111,172.189,49.188,159.810
C02400=1022.662,372.455,-147.151,172.197,49.187,159.812
C02401=1022.670,372.702,-147.192,172.206,49.187,159.813
C02402=1022.679,372.948,-147.232,172.214,49.187,159.814
C02403=1022.687,373.195,-147.272,172.224,49.187,159.816
C02404=1022.696,373.442,-147.312,172.232,49.187,159.817
C02405=1022.704,373.688,-147.353,172.241,49.188,159.818
C02406=1022.713,373.935,-147.393,172.249,49.188,159.820
C02407=1022.721,374.181,-147.434,172.258,49.188,159.821
C02408=1022.730,374.427,-147.474,172.267,49.188,159.823
C02409=1022.739,374.675,-147.514,172.275,49.188,159.824
C02410=1022.747,374.921,-147.554,172.284,49.188,159.825
C02411=1022.756,375.168,-147.595,172.292,49.188,159.827
C02412=1022.765,375.414,-147.635,172.302,49.188,159.828
C02413=1022.773,375.661,-147.676,172.310,49.188,159.829
C02414=1022.783,375.907,-147.716,172.319,49.188,159.831
C02415=1022.791,376.154,-147.757,172.328,49.189,159.832
C02416=1022.799,376.401,-147.798,172.337,49.189,159.834
C02417=1022.808,376.646,-147.838,172.345,49.189,159.835
C02418=1022.817,376.893,-147.880,172.354,49.189,159.836
C02419=1022.825,377.139,-147.920,172.364,49.189,159.838
C02420=1022.834,377.386,-147.961,172.372,49.189,159.839
C02421=1022.843,377.632,-148.003,172.381,49.190,159.841
C02422=1022.851,377.879,-148.044,172.390,49.190,159.842
C02423=1022.860,378.125,-148.084,172.399,49.191,159.844
C02424=1022.869,378.372,-148.126,172.408,49.191,159.845
C02425=1022.877,378.618,-148.167,172.418,49.191,159.847
C02426=1022.886,378.864,-148.208,172.426,49.191,159.848
C02427=1022.895,379.111,-148.249,172.435,49.192,159.850
C02428=1022.903,379.357,-148.291,172.444,49.192,159.851
C02429=1022.912,379.603,-148.332,172.453,49.193,159.853
C02430=1022.921,379.850,-148.373,172.462,49.193,159.854
C02431=1022.930,380.096,-148.414,172.471,49.193,159.856
C02432=1022.938,380.342,-148.456,172.480,49.194,159.857
C02433=1022.947,380.589,-148.497,172.490,49.194,159.859
C02434=1022.957,380.847,-148.540,172.500,49.195,159.860
C02435=1022.965,381.105,-148.584,172.509,49.195,159.862
C02436=1022.975,381.364,-148.627,172.519,49.196,159.864
C02437=1022.984,381.622,-148.671,172.528,49.196,159.865
C02438=1022.993,381.868,-148.712,172.538,49.197,159.867
C02439=1023.003,382.114,-148.754,172.547,49.197,159.868
C02440=1023.012,382.360,-148.795,172.557,49.198,159.870
C02441=1023.021,382.607,-148.837,172.566,49.198,159.872
C02442=1023.030,382.853,-148.879,172.575,49.199,159.873
C02443=1023.039,383.100,-148.920,172.584,49.200,159.875
C02444=1023.048,383.346,-148.962,172.594,49.200,159.876
C02445=1023.056,383.592,-149.004,172.603,49.201,159.878
C02446=1023.066,383.838,-149.045,172.613,49.201,159.880
C02447=1023.075,384.085,-149.087,172.623,49.201,159.881
C02448=1023.084,384.331,-149.128,172.631,49.202,159.883
C02449=1023.093,384.577,-149.170,172.641,49.202,159.884
C02450=1023.102,384.823,-149.213,172.650,49.203,159.886
C02451=1023.111,385.070,-149.254,172.660,49.204,159.888
C02452=1023.120,385.316,-149.296,172.670,49.204,159.889
C02453=1023.130,385.562,-149.339,172.679,49.205,159.891
C02454=1023.140,385.808,-149.380,172.689,49.206,159.893
C02455=1023.149,386.055,-149.422,172.699,49.207,159.894
C02456=1023.157,386.301,-149.465,172.708,49.207,159.896
C02457=1023.166,386.547,-149.506,172.718,49.208,159.898
C02458=1023.175,386.793,-149.549,172.728,49.209,159.899
C02459=1023.185,387.039,-149.592,172.737,49.210,159.901
C02460=1023.194,387.286,-149.633,172.747,49.210,159.903
C02461=1023.203,387.531,-149.676,172.757,49.211,159.905
C02462=1023.212,387.777,-149.718,172.767,49.212,159.906
C02463=1023.221,388.025,-149.761,172.776,49.213,159.908
C02464=1023.230,388.270,-149.803,172.786,49.214,159.910
C02465=1023.240,388.517,-149.846,172.796,49.215,159.912
C02466=1023.250,388.763,-149.889,172.806,49.215,159.913
C02467=1023.259,389.008,-149.931,172.816,49.216,159.915
C02468=1023.269,389.255,-149.974,172.825,49.217,159.917
C02469=1023.277,389.501,-150.017,172.836,49.218,159.919
C02470=1023.286,389.747,-150.059,172.846,49.219,159.921
C02471=1023.296,389.993,-150.102,172.856,49.220,159.922
C02472=1023.305,390.239,-150.145,172.866,49.221,159.924
C02473=1023.315,390.485,-150.188,172.876,49.221,159.926
C02474=1023.324,390.731,-150.230,172.885,49.223,159.928
C02475=1023.334,390.978,-150.273,172.896,49.224,159.930
C02476=1023.342,391.223,-150.317,172.906,49.225,159.932
C02477=1023.352,391.470,-150.360,172.916,49.226,159.933
C02478=1023.362,391.715,-150.402,172.926,49.227,159.935
C02479=1023.371,391.961,-150.446,172.936,49.228,159.937
C02480=1023.381,392.208,-150.489,172.947,49.229,159.939
C02481=1023.390,392.454,-150.531,172.957,49.230,159.941
C02482=1023.400,392.699,-150.575,172.967,49.231,159.943
C02483=1023.409,392.946,-150.618,172.977,49.232,159.945
C02484=1023.419,393.191,-150.661,172.988,49.233,159.946
C02485=1023.428,393.438,-150.705,172.998,49.235,159.948
C02486=1023.438,393.684,-150.748,173.008,49.236,159.950
C02487=1023.447,393.929,-150.792,173.019,49.237,159.952
C02488=1023.457,394.176,-150.835,173.029,49.238,159.954
C02489=1023.467,394.422,-150.878,173.039,49.239,159.956
C02490=1023.476,394.668,-150.923,173.050,49.241,159.958
C02491=1023.486,394.913,-150.966,173.060,49.242,159.960
C02492=1023.495,395.159,-151.010,173.071,49.243,159.962
C02493=1023.505,395.405,-151.053,173.081,49.244,159.964
C02494=1023.516,395.700,-151.105,173.094,49.246,159.966
C02495=1023.528,395.995,-151.158,173.107,49.247,159.969
C02496=1023.540,396.289,-151.210,173.120,49.249,159.971
C02497=1023.552,396.585,-151.263,173.133,49.250,159.974
C02498=1023.561,396.830,-151.307,173.143,49.252,159.976
C02499=1023.571,397.076,-151.351,173.154,49.253,159.978
C02500=1023.580,397.322,-151.395,173.164,49.255,159.980
C02501=1023.591,397.568,-151.438,173.175,49.256,159.982
C02502=1023.600,397.814,-151.482,173.186,49.257,159.984
C02503=1023.610,398.060,-151.526,173.197,49.258,159.986
C02504=1023.620,398.306,-151.571,173.207,49.260,159.988
C02505=1023.631,398.552,-151.615,173.218,49.262,159.990
C02506=1023.640,398.798,-151.659,173.230,49.263,159.992
C02507=1023.650,399.044,-151.703,173.240,49.264,159.994
C02508=1023.660,399.289,-151.748,173.251,49.266,159.996
C02509=1023.670,399.535,-151.792,173.262,49.267,159.998
C02510=1023.679,399.781,-151.837,173.273,49.269,160.001
C02511=1023.690,400.026,-151.881,173.284,49.270,160.003
C02512=1023.700,400.273,-151.925,173.295,49.272,160.005
C02513=1023.710,400.518,-151.970,173.306,49.274,160.007
C02514=1023.720,400.763,-152.014,173.318,49.275,160.009
C02515=1023.730,401.009,-152.059,173.328,49.276,160.011
C02516=1023.740,401.256,-152.104,173.340,49.278,160.014
C02517=1023.749,401.501,-152.148,173.351,49.279,160.016
C02518=1023.759,401.747,-152.193,173.362,49.281,160.018
C02519=1023.770,401.992,-152.237,173.374,49.283,160.020
C02520=1023.780,402.238,-152.283,173.384,49.285,160.022
C02521=1023.790,402.484,-152.328,173.396,49.286,160.025
C02522=1023.800,402.729,-152.373,173.407,49.288,160.027
C02523=1023.810,402.975,-152.418,173.419,49.290,160.029
C02524=1023.820,403.220,-152.463,173.430,49.291,160.031
C02525=1023.830,403.467,-152.508,173.442,49.293,160.034
C02526=1023.840,403.712,-152.553,173.454,49.295,160.036
C02527=1023.850,403.958,-152.599,173.464,49.297,160.038
C02528=1023.861,404.203,-152.643,173.476,49.299,160.040
C02529=1023.871,404.449,-152.688,173.487,49.301,160.043
C02530=1023.881,404.694,-152.734,173.499,49.302,160.045
C02531=1023.891,404.940,-152.779,173.511,49.304,160.047
C02532=1023.902,405.186,-152.825,173.522,49.306,160.050
C02533=1023.912,405.431,-152.870,173.534,49.308,160.052
C02534=1023.922,405.677,-152.916,173.546,49.309,160.054
C02535=1023.933,405.923,-152.961,173.558,49.311,160.057
C02536=1023.943,406.168,-153.006,173.569,49.314,160.059
C02537=1023.954,406.413,-153.052,173.581,49.315,160.061
C02538=1023.964,406.660,-153.097,173.593,49.317,160.064
C02539=1023.975,406.905,-153.143,173.605,49.319,160.066
C02540=1023.985,407.150,-153.188,173.617,49.321,160.069
C02541=1023.996,407.396,-153.234,173.628,49.323,160.071
C02542=1024.006,407.641,-153.280,173.640,49.325,160.073
C02543=1024.017,407.887,-153.326,173.652,49.327,160.076
C02544=1024.027,408.133,-153.371,173.665,49.329,160.078
C02545=1024.039,408.378,-153.417,173.677,49.331,160.081
C02546=1024.049,408.624,-153.463,173.689,49.333,160.083
C02547=1024.060,408.869,-153.508,173.701,49.335,160.086
C02548=1024.071,409.114,-153.555,173.713,49.337,160.088
C02549=1024.081,409.360,-153.601,173.725,49.339,160.091
C02550=1024.092,409.606,-153.647,173.738,49.341,160.093
C02551=1024.103,409.851,-153.693,173.750,49.343,160.096
C02552=1024.113,410.097,-153.740,173.762,49.346,160.098
C02553=1024.123,410.342,-153.786,173.775,49.348,160.101
C02554=1024.136,410.634,-153.840,173.789,49.350,160.104
C02555=1024.148,410.925,-153.896,173.803,49.353,160.107
C02556=1024.162,411.217,-153.951,173.818,49.356,160.110
C02557=1024.174,411.508,-154.007,173.833,49.358,160.113
C02558=1024.185,411.753,-154.053,173.846,49.360,160.116
C02559=1024.196,411.999,-154.100,173.858,49.363,160.118
C02560=1024.207,412.244,-154.146,173.871,49.365,160.121
C02561=1024.218,412.489,-154.193,173.884,49.367,160.124
C02562=1024.229,412.761,-154.244,173.898,49.370,160.126
C02563=1024.242,413.032,-154.296,173.912,49.373,160.129
C02564=1024.254,413.303,-154.348,173.925,49.375,160.132
C02565=1024.267,413.575,-154.400,173.939,49.378,160.135
C02566=1024.277,413.820,-154.447,173.953,49.380,160.138
C02567=1024.288,414.065,-154.494,173.965,49.383,160.141
C02568=1024.300,414.311,-154.541,173.978,49.385,160.143
C02569=1024.310,414.556,-154.588,173.991,49.387,160.146
C02570=1024.321,414.802,-154.635,174.004,49.390,160.149
C02571=1024.333,415.047,-154.682,174.017,49.392,160.151
C02572=1024.344,415.292,-154.729,174.030,49.394,160.154
C02573=1024.356,415.537,-154.776,174.044,49.397,160.157
C02574=1024.366,415.783,-154.824,174.056,49.400,160.160
C02575=1024.378,416.028,-154.871,174.069,49.402,160.163
C02576=1024.388,416.274,-154.919,174.083,49.405,160.165
C02577=1024.400,416.518,-154.966,174.095,49.407,160.168
C02578=1024.410,416.764,-155.014,174.109,49.410,160.171
C02579=1024.422,417.009,-155.062,174.123,49.412,160.174
C02580=1024.433,417.254,-155.109,174.136,49.415,160.177
C02581=1024.445,417.499,-155.157,174.149,49.418,160.180
C02582=1024.456,417.744,-155.204,174.162,49.420,160.183
C02583=1024.467,417.990,-155.252,174.176,49.423,160.185
C02584=1024.479,418.235,-155.300,174.190,49.426,160.188
C02585=1024.490,418.480,-155.348,174.202,49.428,160.191
C02586=1024.501,418.725,-155.396,174.217,49.431,160.194
C02587=1024.512,418.970,-155.444,174.230,49.434,160.197
C02588=1024.524,419.215,-155.492,174.244,49.436,160.200
C02589=1024.535,419.460,-155.540,174.257,49.439,160.203
C02590=1024.547,419.705,-155.588,174.271,49.442,160.206
C02591=1024.559,419.950,-155.637,174.285,49.445,160.209
C02592=1024.570,420.195,-155.685,174.299,49.448,160.212
C02593=1024.582,420.441,-155.733,174.313,49.450,160.215
C02594=1024.593,420.686,-155.781,174.327,49.453,160.218
C02595=1024.605,420.930,-155.830,174.341,49.456,160.221
C02596=1024.617,421.176,-155.878,174.354,49.459,160.224
C02597=1024.629,421.421,-155.927,174.368,49.462,160.227
C02598=1024.641,421.666,-155.974,174.382,49.465,160.230
C02599=1024.652,421.911,-156.023,174.396,49.468,160.233
C02600=1024.664,422.156,-156.071,174.410,49.471,160.236
C02601=1024.676,422.401,-156.120,174.426,49.474,160.240
C02602=1024.687,422.646,-156.169,174.440,49.476,160.243
C02603=1024.699,422.891,-156.218,174.454,49.479,160.246
C02604=1024.711,423.136,-156.267,174.468,49.483,160.249
C02605=1024.723,423.381,-156.316,174.482,49.486,160.252
C02606=1024.734,423.625,-156.365,174.496,49.488,160.255
C02607=1024.747,423.870,-156.414,174.511,49.492,160.258
C02608=1024.758,424.115,-156.463,174.526,49.495,160.262
C02609=1024.770,424.361,-156.512,174.540,49.498,160.265
C02610=1024.782,424.605,-156.561,174.555,49.501,160.268
C02611=1024.794,424.851,-156.610,174.569,49.504,160.271
C02612=1024.806,425.095,-156.659,174.584,49.507,160.275
C02613=1024.818,425.340,-156.709,174.599,49.510,160.278
C02614=1024.835,425.669,-156.775,174.619,49.515,160.282
C02615=1024.851,425.998,-156.841,174.638,49.519,160.287
C02616=1024.867,426.325,-156.908,174.658,49.523,160.291
C02617=1024.883,426.653,-156.975,174.679,49.528,160.296
C02618=1024.896,426.899,-157.024,174.693,49.531,160.299
C02619=1024.908,427.143,-157.074,174.709,49.534,160.302
C02620=1024.920,427.387,-157.124,174.724,49.537,160.306
C02621=1024.932,427.632,-157.174,174.739,49.541,160.309
C02622=1024.944,427.877,-157.224,174.754,49.544,160.313
C02623=1024.957,428.122,-157.274,174.769,49.548,160.316
C02624=1024.969,428.367,-157.324,174.785,49.551,160.320
C02625=1024.981,428.612,-157.374,174.800,49.554,160.323
C02626=1024.993,428.856,-157.424,174.815,49.558,160.326
C02627=1025.005,429.101,-157.474,174.831,49.561,160.330
C02628=1025.018,429.345,-157.524,174.846,49.565,160.334
C02629=1025.030,429.590,-157.575,174.862,49.568,160.337
C02630=1025.043,429.835,-157.625,174.878,49.571,160.341
C02631=1025.055,430.080,-157.676,174.893,49.575,160.344
C02632=1025.069,430.324,-157.726,174.908,49.579,160.348
C02633=1025.081,430.569,-157.776,174.924,49.582,160.351
C02634=1025.094,430.813,-157.827,174.940,49.586,160.355
C02635=1025.106,431.058,-157.877,174.956,49.590,160.359
C02636=1025.119,431.303,-157.928,174.972,49.593,160.362
C02637=1025.132,431.547,-157.979,174.988,49.597,160.366
C02638=1025.144,431.792,-158.029,175.004,49.600,160.369
C02639=1025.157,432.036,-158.080,175.020,49.604,160.373
C02640=1025.170,432.281,-158.131,175.037,49.607,160.377
C02641=1025.183,432.525,-158.182,175.053,49.611,160.380
C02642=1025.196,432.770,-158.233,175.069,49.615,160.384
C02643=1025.208,433.014,-158.284,175.085,49.619,160.388
C02644=1025.222,433.259,-158.335,175.101,49.622,160.392
C02645=1025.234,433.503,-158.386,175.118,49.626,160.395
C02646=1025.248,433.747,-158.438,175.134,49.630,160.399
C02647=1025.260,433.992,-158.488,175.150,49.634,160.403
C02648=1025.274,434.236,-158.540,175.168,49.637,160.407
C02649=1025.287,434.480,-158.591,175.184,49.641,160.411
C02650=1025.300,434.725,-158.642,175.201,49.645,160.415
C02651=1025.313,434.970,-158.695,175.217,49.649,160.418
C02652=1025.325,435.214,-158.746,175.234,49.652,160.422
C02653=1025.339,435.458,-158.797,175.251,49.656,160.426
C02654=1025.352,435.702,-158.849,175.268,49.660,160.430
C02655=1025.365,435.946,-158.901,175.285,49.664,160.434
C02656=1025.378,436.191,-158.953,175.302,49.668,160.438
C02657=1025.391,436.435,-159.005,175.318,49.672,160.442
C02658=1025.405,436.680,-159.056,175.336,49.676,160.446
C02659=1025.418,436.924,-159.108,175.353,49.680,160.450
C02660=1025.432,437.168,-159.161,175.371,49.684,160.454
C02661=1025.445,437.412,-159.213,175.387,49.689,160.458
C02662=1025.458,437.656,-159.265,175.405,49.692,160.462
C02663=1025.472,437.901,-159.317,175.422,49.696,160.466
C02664=1025.485,438.145,-159.369,175.440,49.700,160.470
C02665=1025.499,438.389,-159.422,175.457,49.704,160.474
C02666=1025.512,438.633,-159.474,175.475,49.708,160.478
C02667=1025.526,438.877,-159.527,175.493,49.712,160.482
C02668=1025.539,439.121,-159.579,175.511,49.717,160.487
C02669=1025.552,439.365,-159.632,175.528,49.721,160.491
C02670=1025.567,439.610,-159.685,175.546,49.725,160.495
C02671=1025.581,439.853,-159.737,175.564,49.730,160.499
C02672=1025.594,440.098,-159.790,175.581,49.734,160.503
C02673=1025.607,440.341,-159.843,175.600,49.738,160.508
C02674=1025.620,440.553,-159.889,175.615,49.741,160.511
C02675=1025.632,440.764,-159.934,175.631,49.745,160.515
C02676=1025.644,440.976,-159.980,175.647,49.749,160.519
C02677=1025.655,441.187,-160.027,175.663,49.753,160.522
C02678=1025.668,441.398,-160.073,175.679,49.756,160.526
C02679=1025.680,441.609,-160.118,175.695,49.760,160.530
C02680=1025.692,441.820,-160.164,175.710,49.764,160.534
C02681=1025.704,442.032,-160.210,175.726,49.768,160.537
C02682=1025.718,442.275,-160.264,175.746,49.772,160.542
C02683=1025.732,442.518,-160.317,175.764,49.777,160.546
C02684=1025.747,442.761,-160.369,175.782,49.781,160.551
C02685=1025.762,443.005,-160.422,175.801,49.785,160.555
C02686=1025.778,443.248,-160.473,175.819,49.789,160.559
C02687=1025.794,443.492,-160.525,175.838,49.794,160.564
C02688=1025.810,443.735,-160.576,175.857,49.798,160.568
C02689=1025.827,443.979,-160.627,175.877,49.801,160.572
C02690=1025.844,444.222,-160.677,175.896,49.805,160.577
C02691=1025.862,444.467,-160.728,175.915,49.809,160.581
C02692=1025.880,444.711,-160.777,175.935,49.813,160.586
C02693=1025.899,444.955,-160.826,175.954,49.817,160.590
C02694=1025.918,445.199,-160.875,175.973,49.820,160.594
C02695=1025.937,445.443,-160.924,175.993,49.823,160.599
C02696=1025.957,445.687,-160.972,176.013,49.827,160.603
C02697=1025.978,445.931,-161.019,176.033,49.830,160.607
C02698=1025.999,446.176,-161.067,176.053,49.834,160.612
C02699=1026.020,446.420,-161.113,176.072,49.837,160.616
C02700=1026.042,446.665,-161.160,176.092,49.840,160.620
C02701=1026.065,446.910,-161.206,176.113,49.843,160.624
C02702=1026.087,447.154,-161.252,176.132,49.847,160.629
C02703=1026.110,447.399,-161.297,176.153,49.849,160.633
C02704=1026.134,447.644,-161.343,176.172,49.852,160.637
C02705=1026.158,447.889,-161.387,176.193,49.855,160.642
C02706=1026.183,448.133,-161.431,176.214,49.858,160.646
C02707=1026.207,448.378,-161.475,176.235,49.861,160.650
C02708=1026.233,448.624,-161.518,176.255,49.864,160.655
C02709=1026.258,448.868,-161.561,176.276,49.866,160.659
C02710=1026.284,449.113,-161.604,176.297,49.869,160.663
C02711=1026.312,449.358,-161.646,176.318,49.872,160.668
C02712=1026.340,449.604,-161.688,176.339,49.874,160.672
C02713=1026.367,449.849,-161.729,176.361,49.876,160.676
C02714=1026.395,450.095,-161.770,176.381,49.879,160.680
C02715=1026.423,450.340,-161.811,176.402,49.881,160.684
C02716=1026.452,450.585,-161.851,176.424,49.883,160.689
C02717=1026.482,450.831,-161.891,176.446,49.886,160.693
C02718=1026.512,451.076,-161.931,176.468,49.887,160.697
C02719=1026.543,451.322,-161.970,176.489,49.889,160.702
C02720=1026.573,451.567,-162.009,176.511,49.892,160.706
C02721=1026.605,451.812,-162.047,176.533,49.893,160.710
C02722=1026.637,452.059,-162.084,176.555,49.895,160.714
C02723=1026.669,452.305,-162.123,176.577,49.897,160.719
C02724=1026.702,452.550,-162.160,176.600,49.899,160.723
C02725=1026.734,452.795,-162.196,176.622,49.901,160.727
C02726=1026.769,453.041,-162.232,176.644,49.903,160.732
C02727=1026.803,453.287,-162.269,176.667,49.904,160.736
C02728=1026.838,453.533,-162.304,176.689,49.906,160.740
C02729=1026.872,453.778,-162.340,176.711,49.908,160.744
C02730=1026.908,454.024,-162.374,176.735,49.909,160.749
C02731=1026.944,454.271,-162.409,176.757,49.910,160.753
C02732=1026.981,454.516,-162.442,176.780,49.912,160.757
C02733=1027.017,454.762,-162.476,176.803,49.913,160.762
C02734=1026.744,454.840,-162.814,176.805,49.972,160.781
C02735=1026.707,454.594,-162.781,176.783,49.971,160.777
C02736=1026.671,454.349,-162.748,176.760,49.970,160.772
C02737=1026.635,454.103,-162.713,176.736,49.968,160.768
C02738=1026.599,453.856,-162.678,176.714,49.967,160.764
C02739=1026.564,453.611,-162.643,176.691,49.966,160.760
C02740=1026.529,453.366,-162.608,176.668,49.964,160.755
C02741=1026.495,453.119,-162.572,176.646,49.962,160.751
C02742=1026.461,452.873,-162.536,176.624,49.961,160.747
C02743=1026.428,452.628,-162.499,176.601,49.959,160.742
C02744=1026.395,452.382,-162.463,176.579,49.957,160.738
C02745=1026.363,452.137,-162.425,176.556,49.956,160.734
C02746=1026.330,451.890,-162.387,176.534,49.954,160.730
C02747=1026.299,451.645,-162.349,176.513,49.952,160.725
C02748=1026.268,451.401,-162.311,176.490,49.950,160.721
C02749=1026.237,451.154,-162.271,176.469,49.948,160.717
C02750=1026.207,450.909,-162.232,176.447,49.946,160.713
C02751=1026.177,450.664,-162.192,176.425,49.944,160.708
C02752=1026.148,450.418,-162.153,176.404,49.942,160.704
C02753=1026.119,450.173,-162.112,176.382,49.940,160.700
C02754=1026.091,449.927,-162.071,176.361,49.938,160.696
C02755=1026.063,449.682,-162.030,176.340,49.935,160.691
C02756=1026.035,449.437,-161.988,176.319,49.933,160.687
C02757=1026.009,449.192,-161.946,176.298,49.931,160.683
C02758=1025.982,448.947,-161.904,176.277,49.928,160.678
C02759=1025.956,448.701,-161.860,176.256,49.925,160.674
C02760=1025.930,448.456,-161.817,176.235,49.923,160.670
C02761=1025.905,448.211,-161.774,176.214,49.921,160.666
C02762=1025.881,447.967,-161.729,176.194,49.918,160.661
C02763=1025.856,447.722,-161.686,176.173,49.915,160.657
C02764=1025.833,447.477,-161.640,176.152,49.912,160.653
C02765=1025.809,447.232,-161.595,176.133,49.909,160.648
C02766=1025.786,446.987,-161.550,176.112,49.906,160.644
C02767=1025.764,446.743,-161.504,176.091,49.903,160.640
C02768=1025.742,446.498,-161.457,176.072,49.900,160.636
C02769=1025.721,446.254,-161.411,176.052,49.897,160.631
C02770=1025.699,446.009,-161.364,176.032,49.894,160.627
C02771=1025.678,445.765,-161.317,176.012,49.890,160.622
C02772=1025.658,445.520,-161.268,175.992,49.887,160.618
C02773=1025.638,445.276,-161.221,175.972,49.884,160.614
C02774=1025.619,445.032,-161.172,175.953,49.880,160.610
C02775=1025.600,444.788,-161.123,175.933,49.877,160.605
C02776=1025.582,444.544,-161.073,175.914,49.874,160.601
C02777=1025.564,444.301,-161.024,175.895,49.870,160.597
C02778=1025.546,444.056,-160.973,175.876,49.865,160.592
C02779=1025.530,443.812,-160.923,175.856,49.862,160.588
C02780=1025.513,443.569,-160.872,175.837,49.858,160.584
C02781=1025.496,443.325,-160.821,175.818,49.854,160.579
C02782=1025.480,443.082,-160.769,175.799,49.850,160.575
C02783=1025.466,442.838,-160.717,175.780,49.846,160.570
C02784=1025.450,442.595,-160.664,175.762,49.842,160.566
C02785=1025.436,442.352,-160.612,175.744,49.838,160.562
C02786=1025.422,442.109,-160.558,175.725,49.834,160.557
C02787=1025.410,441.901,-160.513,175.709,49.830,160.554
C02788=1025.398,441.694,-160.468,175.694,49.827,160.550
C02789=1025.386,441.488,-160.423,175.678,49.822,160.546
C02790=1025.374,441.280,-160.378,175.662,49.819,160.543
C02791=1025.362,441.073,-160.333,175.646,49.815,160.539
C02792=1025.351,440.866,-160.287,175.631,49.812,160.535
C02793=1025.339,440.659,-160.243,175.615,49.809,160.532
C02794=1025.327,440.452,-160.197,175.601,49.805,160.528
C02795=1025.314,440.208,-160.145,175.583,49.800,160.524
C02796=1025.300,439.964,-160.093,175.564,49.797,160.520
C02797=1025.286,439.721,-160.040,175.546,49.792,160.515
C02798=1025.272,439.476,-159.986,175.528,49.788,160.511
C02799=1025.259,439.232,-159.934,175.511,49.784,160.507
C02800=1025.245,438.988,-159.882,175.493,49.780,160.503
C02801=1025.232,438.744,-159.829,175.475,49.776,160.499
C02802=1025.218,438.500,-159.777,175.458,49.772,160.495
C02803=1025.205,438.256,-159.724,175.440,49.768,160.491
C02804=1025.192,438.011,-159.672,175.423,49.764,160.486
C02805=1025.178,437.766,-159.620,175.405,49.760,160.482
C02806=1025.164,437.523,-159.567,175.387,49.756,160.478
C02807=1025.150,437.279,-159.515,175.370,49.752,160.474
C02808=1025.137,437.035,-159.464,175.352,49.748,160.470
C02809=1025.124,436.791,-159.412,175.335,49.745,160.466
C02810=1025.111,436.546,-159.359,175.319,49.740,160.462
C02811=1025.097,436.302,-159.307,175.301,49.737,160.458
C02812=1025.084,436.058,-159.255,175.284,49.733,160.454
C02813=1025.070,435.813,-159.203,175.267,49.729,160.450
C02814=1025.058,435.569,-159.153,175.250,49.725,160.447
C02815=1025.045,435.324,-159.100,175.233,49.722,160.443
C02816=1025.031,435.080,-159.048,175.217,49.718,160.439
C02817=1025.018,434.835,-158.997,175.200,49.714,160.435
C02818=1025.005,434.592,-158.946,175.183,49.710,160.431
C02819=1024.992,434.347,-158.894,175.166,49.707,160.427
C02820=1024.979,434.103,-158.843,175.150,49.703,160.423
C02821=1024.966,433.858,-158.792,175.133,49.699,160.420
C02822=1024.953,433.614,-158.741,175.116,49.695,160.416
C02823=1024.941,433.370,-158.688,175.100,49.692,160.412
C02824=1024.928,433.125,-158.638,175.083,49.688,160.408
C02825=1024.915,432.880,-158.586,175.067,49.685,160.405
C02826=1024.902,432.636,-158.536,175.051,49.681,160.401
C02827=1024.889,432.391,-158.484,175.034,49.678,160.397
C02828=1024.876,432.147,-158.434,175.018,49.674,160.393
C02829=1024.863,431.903,-158.384,175.002,49.670,160.390
C02830=1024.850,431.658,-158.333,174.986,49.667,160.386
C02831=1024.837,431.413,-158.282,174.971,49.663,160.383
C02832=1024.825,431.169,-158.231,174.955,49.660,160.379
C02833=1024.812,430.924,-158.181,174.938,49.657,160.375
C02834=1024.799,430.680,-158.130,174.922,49.653,160.372
C02835=1024.787,430.435,-158.080,174.906,49.650,160.368
C02836=1024.774,430.191,-158.029,174.890,49.646,160.365
C02837=1024.762,429.946,-157.979,174.876,49.642,160.361
C02838=1024.749,429.702,-157.928,174.860,49.639,160.357
C02839=1024.736,429.457,-157.879,174.844,49.636,160.354
C02840=1024.724,429.212,-157.829,174.828,49.633,160.350
C02841=1024.712,428.967,-157.779,174.813,49.629,160.347
C02842=1024.699,428.723,-157.728,174.797,49.626,160.344
C02843=1024.687,428.478,-157.678,174.781,49.623,160.340
C02844=1024.674,428.234,-157.628,174.767,49.619,160.337
C02845=1024.662,427.989,-157.577,174.751,49.616,160.333
C02846=1024.650,427.744,-157.527,174.736,49.613,160.330
C02847=1024.638,427.499,-157.478,174.721,49.609,160.326
C02848=1024.626,427.254,-157.428,174.706,49.607,160.323
C02849=1024.614,427.009,-157.378,174.690,49.603,160.319
C02850=1024.601,426.765,-157.328,174.675,49.600,160.316
C02851=1024.586,426.434,-157.262,174.655,49.595,160.312
C02852=1024.569,426.104,-157.194,174.634,49.592,160.307
C02853=1024.552,425.773,-157.128,174.614,49.587,160.303
C02854=1024.536,425.441,-157.060,174.595,49.583,160.298
C02855=1024.524,425.197,-157.011,174.580,49.580,160.295
C02856=1024.512,424.952,-156.962,174.565,49.577,160.292
C02857=1024.500,424.707,-156.913,174.551,49.574,160.289
C02858=1024.488,424.462,-156.864,174.536,49.571,160.285
C02859=1024.476,424.217,-156.815,174.521,49.568,160.282
C02860=1024.464,423.973,-156.765,174.507,49.565,160.279
C02861=1024.452,423.728,-156.717,174.492,49.562,160.276
C02862=1024.440,423.483,-156.667,174.478,49.558,160.272
C02863=1024.429,423.238,-156.618,174.463,49.556,160.269
C02864=1024.417,422.993,-156.570,174.449,49.553,160.266
C02865=1024.405,422.747,-156.521,174.434,49.550,160.263
C02866=1024.393,422.503,-156.472,174.420,49.547,160.260
C02867=1024.381,422.258,-156.424,174.406,49.544,160.257
C02868=1024.369,422.013,-156.374,174.392,49.541,160.254
C02869=1024.358,421.767,-156.326,174.378,49.538,160.251
C02870=1024.346,421.523,-156.278,174.363,49.536,160.247
C02871=1024.335,421.278,-156.229,174.349,49.533,160.244
C02872=1024.323,421.033,-156.181,174.335,49.530,160.241
C02873=1024.311,420.787,-156.132,174.321,49.527,160.238
C02874=1024.299,420.542,-156.084,174.307,49.525,160.235
C02875=1024.288,420.297,-156.035,174.293,49.522,160.232
C02876=1024.276,420.052,-155.988,174.280,49.519,160.229
C02877=1024.265,419.807,-155.939,174.266,49.517,160.226
C02878=1024.253,419.562,-155.892,174.252,49.514,160.223
C02879=1024.242,419.317,-155.843,174.239,49.511,160.220
C02880=1024.230,419.071,-155.796,174.224,49.509,160.217
C02881=1024.218,418.826,-155.748,174.211,49.506,160.215
C02882=1024.207,418.581,-155.700,174.197,49.503,160.211
C02883=1024.195,418.336,-155.652,174.184,49.501,160.209
C02884=1024.185,418.091,-155.604,174.170,49.498,160.206
C02885=1024.173,417.846,-155.556,174.156,49.495,160.203
C02886=1024.162,417.601,-155.508,174.143,49.493,160.200
C02887=1024.150,417.356,-155.460,174.130,49.490,160.197
C02888=1024.139,417.110,-155.413,174.116,49.488,160.194
C02889=1024.128,416.866,-155.366,174.103,49.485,160.192
C02890=1024.117,416.620,-155.317,174.090,49.483,160.189
C02891=1024.105,416.374,-155.270,174.076,49.481,160.186
C02892=1024.095,416.130,-155.222,174.063,49.478,160.183
C02893=1024.083,415.884,-155.175,174.050,49.476,160.180
C02894=1024.073,415.640,-155.127,174.037,49.473,160.177
C02895=1024.061,415.394,-155.080,174.023,49.471,160.175
C02896=1024.050,415.148,-155.033,174.011,49.468,160.172
C02897=1024.039,414.903,-154.987,173.997,49.466,160.169
C02898=1024.028,414.658,-154.938,173.985,49.463,160.166
C02899=1024.016,414.412,-154.891,173.971,49.462,160.164
C02900=1024.005,414.167,-154.845,173.959,49.459,160.161
C02901=1023.994,413.921,-154.798,173.946,49.457,160.158
C02902=1023.984,413.676,-154.751,173.933,49.454,160.156
C02903=1023.973,413.431,-154.704,173.920,49.452,160.153
C02904=1023.961,413.186,-154.657,173.908,49.449,160.150
C02905=1023.950,412.941,-154.610,173.894,49.448,160.148
C02906=1023.940,412.695,-154.565,173.882,49.445,160.145
C02907=1023.929,412.449,-154.517,173.870,49.443,160.142
C02908=1023.918,412.204,-154.470,173.856,49.441,160.140
C02909=1023.907,411.959,-154.424,173.844,49.439,160.137
C02910=1023.896,411.713,-154.377,173.831,49.436,160.134
C02911=1023.882,411.394,-154.316,173.815,49.434,160.131
C02912=1023.867,411.074,-154.256,173.798,49.431,160.128
C02913=1023.854,410.755,-154.195,173.782,49.428,160.124
C02914=1023.840,410.434,-154.135,173.766,49.425,160.121
C02915=1023.830,410.189,-154.089,173.754,49.423,160.118
C02916=1023.819,409.944,-154.043,173.741,49.421,160.116
C02917=1023.808,409.699,-153.996,173.729,49.419,160.114
C02918=1023.798,409.453,-153.950,173.717,49.417,160.111
C02919=1023.787,409.207,-153.904,173.705,49.415,160.108
C02920=1023.776,408.962,-153.858,173.693,49.413,160.106
C02921=1023.765,408.716,-153.812,173.681,49.411,160.103
C02922=1023.755,408.471,-153.766,173.669,49.410,160.101
C02923=1023.744,408.225,-153.721,173.656,49.407,160.099
C02924=1023.734,407.979,-153.675,173.644,49.406,160.096
C02925=1023.723,407.734,-153.629,173.632,49.403,160.094
C02926=1023.712,407.488,-153.583,173.620,49.402,160.091
C02927=1023.701,407.243,-153.538,173.608,49.400,160.089
C02928=1023.691,406.998,-153.492,173.596,49.398,160.086
C02929=1023.681,406.752,-153.447,173.584,49.396,160.084
C02930=1023.670,406.506,-153.401,173.573,49.394,160.082
C02931=1023.659,406.261,-153.355,173.561,49.393,160.079
C02932=1023.650,406.015,-153.310,173.549,49.390,160.077
C02933=1023.639,405.770,-153.264,173.537,49.389,160.075
C02934=1023.628,405.524,-153.218,173.525,49.387,160.072
C02935=1023.619,405.278,-153.174,173.513,49.385,160.070
C02936=1023.607,405.033,-153.128,173.502,49.383,160.068
C02937=1023.597,404.787,-153.083,173.490,49.382,160.065
C02938=1023.587,404.541,-153.038,173.478,49.380,160.063
C02939=1023.570,404.134,-152.962,173.459,49.377,160.059
C02940=1023.553,403.727,-152.888,173.441,49.374,160.055
C02941=1023.537,403.320,-152.813,173.421,49.372,160.052
C02942=1023.520,402.913,-152.739,173.402,49.369,160.048
C02943=1023.509,402.668,-152.693,173.390,49.368,160.046
C02944=1023.499,402.422,-152.648,173.380,49.366,160.043
C02945=1023.490,402.177,-152.604,173.368,49.365,160.041
C02946=1023.479,401.930,-152.558,173.357,49.362,160.039
C02947=1023.470,401.685,-152.514,173.345,49.361,160.037
C02948=1023.459,401.440,-152.469,173.335,49.359,160.035
C02949=1023.450,401.194,-152.425,173.323,49.358,160.032
C02950=1023.440,400.947,-152.380,173.312,49.356,160.030
C02951=1023.430,400.702,-152.335,173.300,49.355,160.028
C02952=1023.419,400.457,-152.291,173.290,49.354,160.026
C02953=1023.410,400.211,-152.246,173.278,49.352,160.024
C02954=1023.400,399.964,-152.202,173.267,49.350,160.022
C02955=1023.389,399.719,-152.158,173.256,49.349,160.020
C02956=1023.379,399.474,-152.113,173.245,49.348,160.017
C02957=1023.370,399.227,-152.069,173.235,49.346,160.015
C02958=1023.360,398.982,-152.024,173.223,49.345,160.013
C02959=1023.350,398.736,-151.980,173.213,49.344,160.011
C02960=1023.341,398.490,-151.936,173.202,49.342,160.009
C02961=1023.330,398.245,-151.892,173.190,49.341,160.007
C02962=1023.321,397.999,-151.848,173.180,49.340,160.005
C02963=1023.311,397.753,-151.804,173.169,49.338,160.003
C02964=1023.301,397.507,-151.759,173.158,49.337,160.001
C02965=1023.291,397.261,-151.716,173.147,49.336,159.999
C02966=1023.281,397.015,-151.672,173.137,49.334,159.997
C02967=1023.266,396.633,-151.603,173.120,49.333,159.994
C02968=1023.250,396.252,-151.536,173.103,49.330,159.990
C02969=1023.236,395.870,-151.468,173.086,49.329,159.987
C02970=1023.221,395.488,-151.400,173.071,49.327,159.984
C02971=1023.211,395.243,-151.357,173.059,49.326,159.982
C02972=1023.202,394.997,-151.313,173.049,49.325,159.980
C02973=1023.192,394.751,-151.269,173.038,49.323,159.978
C02974=1023.182,394.505,-151.226,173.028,49.322,159.976
C02975=1023.172,394.259,-151.182,173.018,49.322,159.975
C02976=1023.163,394.014,-151.139,173.007,49.320,159.973
C02977=1023.153,393.767,-151.095,172.997,49.319,159.971
C02978=1023.144,393.521,-151.052,172.987,49.318,159.969
C02979=1023.135,393.276,-151.008,172.975,49.317,159.967
C02980=1023.125,393.029,-150.966,172.965,49.316,159.965
C02981=1023.116,392.783,-150.922,172.955,49.315,159.963
C02982=1023.106,392.537,-150.879,172.945,49.314,159.961
C02983=1023.096,392.291,-150.836,172.934,49.313,159.959
C02984=1023.086,392.045,-150.793,172.924,49.312,159.957
C02985=1023.078,391.799,-150.750,172.914,49.311,159.955
C02986=1023.068,391.553,-150.706,172.904,49.310,159.954
C02987=1023.058,391.307,-150.664,172.893,49.309,159.952
C02988=1023.049,391.061,-150.620,172.883,49.308,159.950
C02989=1023.040,390.815,-150.578,172.873,49.307,159.948
C02990=1023.030,390.569,-150.535,172.863,49.306,159.946
C02991=1023.021,390.323,-150.492,172.853,49.306,159.945
C02992=1023.012,390.076,-150.449,172.844,49.305,159.943
C02993=1023.002,389.831,-150.406,172.834,49.304,159.941
C02994=1022.992,389.584,-150.363,172.823,49.303,159.939
C02995=1022.983,389.339,-150.321,172.813,49.302,159.937
C02996=1022.975,389.092,-150.278,172.803,49.302,159.936
C02997=1022.965,388.846,-150.235,172.793,49.301,159.934
C02998=1022.956,388.600,-150.193,172.783,49.300,159.932
C02999=1022.947,388.354,-150.151,172.773,49.299,159.930
C03000=1022.937,388.107,-150.108,172.764,49.298,159.929
C03001=1022.928,387.861,-150.065,172.754,49.297,159.927
C03002=1022.919,387.616,-150.023,172.744,49.297,159.925
C03003=1022.910,387.369,-149.981,172.734,49.296,159.923
C03004=1022.900,387.123,-149.938,172.724,49.296,159.922
C03005=1022.891,386.877,-149.896,172.715,49.295,159.920
C03006=1022.882,386.631,-149.854,172.705,49.294,159.918
C03007=1022.872,386.384,-149.811,172.695,49.294,159.917
C03008=1022.863,386.138,-149.770,172.685,49.293,159.915
C03009=1022.854,385.892,-149.727,172.676,49.292,159.913
C03010=1022.845,385.646,-149.685,172.666,49.292,159.912
C03011=1022.836,385.399,-149.644,172.656,49.291,159.910
C03012=1022.827,385.154,-149.601,172.646,49.290,159.908
C03013=1022.818,384.907,-149.559,172.637,49.290,159.907
C03014=1022.809,384.660,-149.518,172.628,49.289,159.905
C03015=1022.800,384.414,-149.476,172.618,49.289,159.903
C03016=1022.790,384.168,-149.433,172.609,49.288,159.902
C03017=1022.781,383.922,-149.392,172.599,49.288,159.900
C03018=1022.772,383.676,-149.351,172.589,49.287,159.898
C03019=1022.763,383.429,-149.309,172.580,49.287,159.897
C03020=1022.754,383.183,-149.267,172.571,49.286,159.895
C03021=1022.745,382.937,-149.225,172.561,49.286,159.894
C03022=1022.736,382.690,-149.184,172.552,49.285,159.892
C03023=1022.727,382.444,-149.142,172.542,49.285,159.890
C03024=1022.718,382.198,-149.100,172.534,49.285,159.889
C03025=1022.709,381.952,-149.059,172.524,49.284,159.887
C03026=1022.700,381.705,-149.017,172.515,49.284,159.886
C03027=1022.691,381.444,-148.974,172.505,49.283,159.884
C03028=1022.681,381.184,-148.930,172.495,49.283,159.883
C03029=1022.672,380.924,-148.886,172.486,49.283,159.881
C03030=1022.662,380.664,-148.843,172.476,49.282,159.879
C03031=1022.654,380.418,-148.801,172.466,49.282,159.878
C03032=1022.645,380.171,-148.760,172.457,49.282,159.876
C03033=1022.636,379.925,-148.719,172.448,49.281,159.875
C03034=1022.627,379.678,-148.677,172.439,49.281,159.873
C03035=1022.619,379.432,-148.636,172.429,49.281,159.872
C03036=1022.609,379.186,-148.595,172.421,49.281,159.870
C03037=1022.601,378.939,-148.554,172.411,49.280,159.869
C03038=1022.592,378.693,-148.512,172.403,49.280,159.867
C03039=1022.584,378.446,-148.472,172.394,49.279,159.866
C03040=1022.575,378.200,-148.430,172.384,49.280,159.864
C03041=1022.566,377.953,-148.389,172.375,49.279,159.863
C03042=1022.558,377.707,-148.348,172.366,49.279,159.861
C03043=1022.549,377.461,-148.307,172.357,49.279,159.860
C03044=1022.541,377.214,-148.267,172.349,49.278,159.858
C03045=1022.532,376.967,-148.226,172.339,49.279,159.857
C03046=1022.524,376.722,-148.184,172.331,49.278,159.856
C03047=1022.515,376.475,-148.143,172.322,49.278,159.854
C03048=1022.506,376.228,-148.103,172.312,49.278,159.853
C03049=1022.498,375.982,-148.062,172.304,49.278,159.851
C03050=1022.488,375.735,-148.022,172.295,49.278,159.850
C03051=1022.480,375.489,-147.981,172.286,49.278,159.849
C03052=1022.472,375.242,-147.940,172.278,49.278,159.847
C03053=1022.463,374.996,-147.900,172.269,49.278,159.846
C03054=1022.454,374.749,-147.859,172.260,49.278,159.844
C03055=1022.445,374.503,-147.819,172.251,49.278,159.843
C03056=1022.437,374.255,-147.779,172.243,49.278,159.842
C03057=1022.428,374.009,-147.739,172.233,49.278,159.840
C03058=1022.420,373.762,-147.698,172.225,49.278,159.839
C03059=1022.411,373.516,-147.658,172.217,49.278,159.838
C03060=1022.403,373.269,-147.618,172.208,49.278,159.836
C03061=1022.394,373.023,-147.577,172.199,49.278,159.835
C03062=1022.386,372.776,-147.537,172.190,49.278,159.834
C03063=1022.377,372.530,-147.497,172.182,49.278,159.832
C03064=1022.369,372.283,-147.456,172.174,49.278,159.831
C03065=1022.360,372.037,-147.416,172.165,49.278,159.830
C03066=1022.352,371.790,-147.377,172.156,49.278,159.828
C03067=1022.343,371.543,-147.336,172.148,49.279,159.827
C03068=1022.335,371.296,-147.296,172.139,49.279,159.826
C03069=1022.326,371.050,-147.256,172.131,49.279,159.825
C03070=1022.319,370.803,-147.216,172.123,49.279,159.823
C03071=1022.310,370.557,-147.176,172.114,49.279,159.822
C03072=1022.302,370.310,-147.136,172.105,49.280,159.821
C03073=1022.293,370.063,-147.097,172.097,49.280,159.819
C03074=1022.285,369.817,-147.056,172.089,49.280,159.818
C03075=1022.277,369.570,-147.017,172.080,49.280,159.817
C03076=1022.269,369.323,-146.977,172.072,49.280,159.816
C03077=1022.260,369.078,-146.937,172.063,49.280,159.814
C03078=1022.252,368.831,-146.897,172.055,49.281,159.813
C03079=1022.243,368.583,-146.857,172.047,49.281,159.812
C03080=1022.236,368.336,-146.817,172.039,49.281,159.811
C03081=1022.227,368.090,-146.778,172.031,49.281,159.810
C03082=1022.219,367.843,-146.739,172.022,49.282,159.808
C03083=1022.211,367.601,-146.700,172.014,49.282,159.807
C03084=1022.202,367.359,-146.661,172.006,49.282,159.806
C03085=1022.194,367.116,-146.622,171.998,49.283,159.805
C03086=1022.186,366.874,-146.583,171.990,49.283,159.804
C03087=1022.178,366.631,-146.544,171.982,49.284,159.803
C03088=1022.169,366.389,-146.506,171.974,49.284,159.801
C03089=1022.162,366.145,-146.468,171.965,49.285,159.800
C03090=1022.154,365.903,-146.429,171.957,49.285,159.799
C03091=1022.146,365.657,-146.390,171.949,49.285,159.798
C03092=1022.137,365.410,-146.350,171.941,49.286,159.797
C03093=1022.129,365.163,-146.311,171.933,49.286,159.796
C03094=1022.121,364.916,-146.272,171.925,49.287,159.794
C03095=1022.112,364.670,-146.233,171.917,49.287,159.793
C03096=1022.105,364.423,-146.193,171.909,49.288,159.792
C03097=1022.097,364.176,-146.155,171.901,49.288,159.791
C03098=1022.089,363.930,-146.116,171.893,49.289,159.790
C03099=1022.080,363.682,-146.077,171.885,49.290,159.789
C03100=1022.072,363.436,-146.038,171.877,49.290,159.788
C03101=1022.064,363.189,-145.999,171.869,49.291,159.787
C03102=1022.055,362.942,-145.960,171.861,49.291,159.785
C03103=1022.048,362.695,-145.921,171.853,49.292,159.785
C03104=1022.040,362.449,-145.881,171.845,49.293,159.783
C03105=1022.032,362.201,-145.843,171.838,49.293,159.782
C03106=1022.024,361.954,-145.804,171.829,49.293,159.781
C03107=1022.016,361.708,-145.765,171.822,49.294,159.780
C03108=1022.008,361.461,-145.727,171.814,49.295,159.779
C03109=1022.000,361.213,-145.688,171.805,49.295,159.778
C03110=1021.992,360.968,-145.649,171.798,49.296,159.777
C03111=1021.984,360.720,-145.610,171.790,49.297,159.776
C03112=1021.976,360.473,-145.571,171.783,49.297,159.775
C03113=1021.969,360.227,-145.533,171.775,49.298,159.774
C03114=1021.960,359.980,-145.494,171.767,49.299,159.773
C03115=1021.953,359.734,-145.456,171.759,49.299,159.772
C03116=1021.944,359.486,-145.417,171.751,49.300,159.771
C03117=1021.936,359.239,-145.378,171.743,49.301,159.770
C03118=1021.929,358.993,-145.340,171.735,49.302,159.769
C03119=1021.921,358.745,-145.301,171.729,49.303,159.768
C03120=1021.913,358.499,-145.263,171.720,49.303,159.767
C03121=1021.905,358.251,-145.225,171.713,49.304,159.766
C03122=1021.898,358.005,-145.187,171.705,49.305,159.765
C03123=1021.890,357.757,-145.148,171.697,49.306,159.764
C03124=1021.881,357.511,-145.111,171.690,49.306,159.763
C03125=1021.873,357.264,-145.072,171.682,49.307,159.762
C03126=1021.866,357.017,-145.035,171.675,49.308,159.761
C03127=1021.858,356.770,-144.996,171.667,49.309,159.760
C03128=1021.850,356.523,-144.958,171.659,49.310,159.759
C03129=1021.842,356.276,-144.919,171.652,49.311,159.758
C03130=1021.834,356.029,-144.882,171.644,49.312,159.757
C03131=1021.826,355.782,-144.844,171.637,49.313,159.756
C03132=1021.818,355.535,-144.805,171.629,49.314,159.755
C03133=1021.810,355.287,-144.768,171.622,49.315,159.754
C03134=1021.803,355.041,-144.729,171.614,49.316,159.753
C03135=1021.796,354.794,-144.692,171.607,49.317,159.752
C03136=1021.787,354.547,-144.654,171.599,49.318,159.751
C03137=1021.780,354.300,-144.616,171.592,49.318,159.750
C03138=1021.772,354.053,-144.578,171.584,49.319,159.749
C03139=1021.764,353.805,-144.540,171.577,49.321,159.748
C03140=1021.756,353.559,-144.503,171.570,49.321,159.748
C03141=1021.749,353.312,-144.465,171.562,49.322,159.747
C03142=1021.740,353.064,-144.428,171.555,49.324,159.746
C03143=1021.734,352.826,-144.392,171.548,49.325,159.745
C03144=1021.726,352.587,-144.354,171.540,49.326,159.744
C03145=1021.718,352.348,-144.319,171.534,49.326,159.743
C03146=1021.711,352.109,-144.282,171.526,49.328,159.742
C03147=1021.703,351.870,-144.246,171.519,49.329,159.742
C03148=1021.696,351.631,-144.209,171.512,49.330,159.741
C03149=1021.688,351.392,-144.174,171.505,49.331,159.740
C03150=1021.681,351.152,-144.137,171.498,49.332,159.739
C03151=1021.674,350.905,-144.100,171.491,49.334,159.738
C03152=1021.666,350.658,-144.063,171.483,49.335,159.737
C03153=1021.659,350.411,-144.025,171.477,49.335,159.736
C03154=1021.650,350.164,-143.988,171.469,49.337,159.736
C03155=1021.643,349.916,-143.950,171.461,49.338,159.735
C03156=1021.635,349.669,-143.913,171.455,49.339,159.734
C03157=1021.627,349.422,-143.876,171.447,49.341,159.733
C03158=1021.620,349.175,-143.838,171.440,49.342,159.732
C03159=1021.613,348.928,-143.801,171.433,49.343,159.731
C03160=1021.605,348.681,-143.764,171.425,49.344,159.731
C03161=1021.598,348.434,-143.726,171.419,49.345,159.730
C03162=1021.590,348.187,-143.689,171.412,49.347,159.729
C03163=1021.583,347.940,-143.652,171.404,49.348,159.728
C03164=1021.575,347.693,-143.616,171.398,49.349,159.727
C03165=1021.568,347.446,-143.578,171.390,49.350,159.727
C03166=1021.560,347.199,-143.541,171.383,49.352,159.726
C03167=1021.553,346.951,-143.504,171.376,49.353,159.725
C03168=1021.545,346.704,-143.467,171.370,49.355,159.724
C03169=1021.537,346.457,-143.431,171.362,49.356,159.723
C03170=1021.530,346.210,-143.394,171.355,49.357,159.723
C03171=1021.522,345.963,-143.357,171.348,49.359,159.722
C03172=1021.515,345.715,-143.320,171.341,49.360,159.721
C03173=1021.507,345.468,-143.283,171.334,49.362,159.721
C03174=1021.499,345.221,-143.247,171.327,49.363,159.720
C03175=1021.492,344.974,-143.209,171.320,49.364,159.719
C03176=1021.485,344.727,-143.173,171.313,49.366,159.718
C03177=1021.477,344.480,-143.137,171.306,49.367,159.718
C03178=1021.470,344.232,-143.100,171.299,49.369,159.717
C03179=1021.462,343.985,-143.063,171.293,49.370,159.716
C03180=1021.454,343.738,-143.027,171.285,49.372,159.715
C03181=1021.447,343.490,-142.990,171.279,49.373,159.715
C03182=1021.440,343.244,-142.954,171.272,49.375,159.714
C03183=1021.432,342.997,-142.917,171.265,49.376,159.713
C03184=1021.425,342.749,-142.880,171.258,49.378,159.712
C03185=1021.418,342.502,-142.844,171.251,49.379,159.712
C03186=1021.410,342.254,-142.808,171.244,49.381,159.711
C03187=1021.404,342.007,-142.771,171.238,49.382,159.710
C03188=1021.396,341.760,-142.734,171.230,49.384,159.710
C03189=1021.388,341.513,-142.698,171.224,49.385,159.709
C03190=1021.381,341.266,-142.662,171.217,49.388,159.708
C03191=1021.374,341.018,-142.625,171.210,49.389,159.708
C03192=1021.366,340.771,-142.589,171.203,49.391,159.707
C03193=1021.359,340.523,-142.553,171.197,49.392,159.706
C03194=1021.352,340.277,-142.517,171.189,49.394,159.706
C03195=1021.345,340.029,-142.480,171.183,49.395,159.705
C03196=1021.338,339.782,-142.445,171.176,49.397,159.704
C03197=1021.330,339.535,-142.408,171.169,49.398,159.704
C03198=1021.322,339.287,-142.372,171.163,49.400,159.703
C03199=1021.315,339.041,-142.336,171.156,49.402,159.702
C03200=1021.308,338.792,-142.301,171.150,49.403,159.702
C03201=1021.300,338.545,-142.265,171.143,49.406,159.701
C03202=1021.293,338.298,-142.229,171.136,49.407,159.700
C03203=1021.287,338.058,-142.194,171.129,49.409,159.700
C03204=1021.279,337.817,-142.159,171.123,49.411,159.699
C03205=1021.272,337.577,-142.123,171.117,49.413,159.699
C03206=1021.265,337.336,-142.089,171.110,49.414,159.698
C03207=1021.258,337.095,-142.054,171.103,49.416,159.698
C03208=1021.250,336.854,-142.019,171.097,49.418,159.697
C03209=1021.243,336.614,-141.985,171.091,49.420,159.696
C03210=1021.237,336.373,-141.950,171.085,49.421,159.696
C03211=1021.229,336.126,-141.914,171.078,49.423,159.695
C03212=1021.222,335.879,-141.878,171.071,49.425,159.694
C03213=1021.215,335.631,-141.842,171.065,49.427,159.694
C03214=1021.208,335.384,-141.807,171.058,49.429,159.693
C03215=1021.201,335.137,-141.771,171.052,49.430,159.693
C03216=1021.193,334.889,-141.736,171.045,49.432,159.692
C03217=1021.186,334.642,-141.700,171.039,49.434,159.692
C03218=1021.179,334.394,-141.664,171.032,49.436,159.691
C03219=1021.172,334.147,-141.629,171.025,49.438,159.690
C03220=1021.165,333.900,-141.593,171.019,49.440,159.690
C03221=1021.158,333.652,-141.558,171.013,49.442,159.689
C03222=1021.151,333.405,-141.522,171.006,49.444,159.689
C03223=1021.144,333.158,-141.487,171.000,49.446,159.688
C03224=1021.137,332.910,-141.451,170.994,49.448,159.688
C03225=1021.129,332.663,-141.416,170.987,49.450,159.687
C03226=1021.122,332.416,-141.381,170.981,49.452,159.687
C03227=1021.115,332.168,-141.346,170.974,49.454,159.686
C03228=1021.108,331.921,-141.310,170.968,49.456,159.686
C03229=1021.101,331.673,-141.275,170.961,49.457,159.685
C03230=1021.093,331.425,-141.240,170.954,49.460,159.684
C03231=1021.086,331.178,-141.205,170.948,49.462,159.684
C03232=1021.079,330.931,-141.169,170.942,49.464,159.683
C03233=1021.072,330.684,-141.134,170.935,49.466,159.683
C03234=1021.064,330.436,-141.099,170.929,49.468,159.682
C03235=1021.057,330.189,-141.064,170.923,49.471,159.682
C03236=1021.051,329.942,-141.029,170.916,49.473,159.682
C03237=1021.044,329.694,-140.994,170.910,49.475,159.681
C03238=1021.036,329.446,-140.960,170.904,49.477,159.681
C03239=1021.029,329.198,-140.925,170.897,49.479,159.680
C03240=1021.023,328.951,-140.889,170.891,49.481,159.680
C03241=1021.015,328.704,-140.855,170.885,49.483,159.679
C03242=1021.008,328.457,-140.820,170.878,49.485,159.678
C03243=1021.002,328.209,-140.785,170.872,49.487,159.678
C03244=1020.995,327.962,-140.750,170.867,49.490,159.678
C03245=1020.987,327.715,-140.715,170.861,49.492,159.677
C03246=1020.980,327.466,-140.680,170.853,49.494,159.677
C03247=1020.973,327.219,-140.645,170.847,49.496,159.676
C03248=1020.967,326.971,-140.610,170.842,49.499,159.676
C03249=1020.959,326.724,-140.575,170.835,49.501,159.675
C03250=1020.953,326.476,-140.541,170.829,49.503,159.675
C03251=1020.945,326.229,-140.506,170.823,49.506,159.675
C03252=1020.938,325.982,-140.473,170.816,49.508,159.674
C03253=1020.931,325.734,-140.437,170.810,49.510,159.674
C03254=1020.924,325.487,-140.404,170.804,49.512,159.673
C03255=1020.916,325.240,-140.369,170.797,49.515,159.673
C03256=1020.909,324.992,-140.335,170.792,49.517,159.672
C03257=1020.903,324.745,-140.300,170.786,49.520,159.672
C03258=1020.895,324.497,-140.266,170.779,49.522,159.672
C03259=1020.888,324.249,-140.232,170.773,49.525,159.671
C03260=1020.881,324.002,-140.197,170.767,49.527,159.671
C03261=1020.874,323.754,-140.164,170.762,49.529,159.670
C03262=1020.867,323.506,-140.130,170.755,49.532,159.670
C03263=1020.860,323.263,-140.095,170.749,49.534,159.670
C03264=1020.853,323.021,-140.062,170.743,49.537,159.669
C03265=1020.846,322.778,-140.028,170.737,49.539,159.669
C03266=1020.839,322.535,-139.996,170.732,49.542,159.669
C03267=1020.832,322.292,-139.961,170.725,49.544,159.668
C03268=1020.825,322.050,-139.928,170.719,49.546,159.668
C03269=1020.819,321.807,-139.894,170.713,49.549,159.667
C03270=1020.812,321.564,-139.862,170.708,49.552,159.667
C03271=1020.804,321.316,-139.828,170.701,49.554,159.667
C03272=1020.798,321.069,-139.793,170.695,49.557,159.666
C03273=1020.791,320.821,-139.759,170.689,49.559,159.666
C03274=1020.783,320.574,-139.725,170.684,49.562,159.666
C03275=1020.777,320.326,-139.691,170.677,49.564,159.665
C03276=1020.770,320.079,-139.657,170.671,49.567,159.665
C03277=1020.763,319.831,-139.623,170.665,49.569,159.665
C03278=1020.756,319.583,-139.589,170.659,49.572,159.664
C03279=1020.749,319.335,-139.555,170.654,49.575,159.664
C03280=1020.743,319.088,-139.521,170.647,49.577,159.664
C03281=1020.736,318.841,-139.488,170.641,49.579,159.663
C03282=1020.728,318.593,-139.454,170.635,49.582,159.663
C03283=1020.722,318.345,-139.419,170.630,49.585,159.662
C03284=1020.715,318.098,-139.386,170.624,49.587,159.662
C03285=1020.708,317.850,-139.352,170.617,49.590,159.662
C03286=1020.702,317.602,-139.318,170.612,49.593,159.662
C03287=1020.695,317.355,-139.284,170.606,49.595,159.661
C03288=1020.688,317.108,-139.250,170.600,49.598,159.661
C03289=1020.681,316.859,-139.217,170.595,49.601,159.661
C03290=1020.675,316.612,-139.183,170.588,49.604,159.660
C03291=1020.668,316.365,-139.149,170.582,49.606,159.660
C03292=1020.661,316.117,-139.116,170.577,49.609,159.660
C03293=1020.654,315.870,-139.082,170.571,49.611,159.659
C03294=1020.648,315.622,-139.048,170.565,49.614,159.659
C03295=1020.641,315.374,-139.015,170.559,49.617,159.659
C03296=1020.634,315.127,-138.981,170.553,49.620,159.658
C03297=1020.628,314.880,-138.948,170.547,49.622,159.658
C03298=1020.621,314.631,-138.914,170.542,49.626,159.658
C03299=1020.614,314.383,-138.880,170.537,49.628,159.658
C03300=1020.608,314.136,-138.847,170.531,49.631,159.657
C03301=1020.600,313.889,-138.813,170.524,49.634,159.657
C03302=1020.595,313.641,-138.780,170.519,49.636,159.657
C03303=1020.588,313.393,-138.746,170.513,49.639,159.657
C03304=1020.581,313.146,-138.713,170.507,49.642,159.656
C03305=1020.574,312.898,-138.679,170.502,49.645,159.656
C03306=1020.568,312.651,-138.645,170.496,49.647,159.656
C03307=1020.562,312.403,-138.612,170.491,49.650,159.656
C03308=1020.555,312.155,-138.579,170.484,49.653,159.655
C03309=1020.549,311.908,-138.546,170.479,49.656,159.655
C03310=1020.541,311.660,-138.512,170.473,49.659,159.655
C03311=1020.536,311.412,-138.479,170.467,49.661,159.654
C03312=1020.529,311.165,-138.445,170.462,49.665,159.654
C03313=1020.522,310.917,-138.412,170.456,49.667,159.654
C03314=1020.516,310.670,-138.379,170.451,49.670,159.654
C03315=1020.510,310.421,-138.345,170.445,49.673,159.654
C03316=1020.503,310.174,-138.311,170.440,49.676,159.653
C03317=1020.497,309.927,-138.279,170.433,49.679,159.653
C03318=1020.489,309.679,-138.246,170.428,49.682,159.653
C03319=1020.483,309.431,-138.213,170.422,49.685,159.653
C03320=1020.476,309.184,-138.181,170.417,49.688,159.653
C03321=1020.469,308.936,-138.148,170.411,49.691,159.652
C03322=1020.462,308.688,-138.115,170.405,49.695,159.652
C03323=1020.456,308.447,-138.083,170.399,49.697,159.652
C03324=1020.450,308.208,-138.052,170.394,49.701,159.652
C03325=1020.442,307.967,-138.020,170.389,49.703,159.652
C03326=1020.436,307.727,-137.989,170.383,49.707,159.651
C03327=1020.429,307.487,-137.957,170.378,49.710,159.651
C03328=1020.423,307.247,-137.925,170.372,49.712,159.651
C03329=1020.416,307.006,-137.893,170.367,49.716,159.651
C03330=1020.409,306.767,-137.862,170.362,49.719,159.651
C03331=1020.403,306.519,-137.829,170.356,49.722,159.651
C03332=1020.397,306.270,-137.797,170.351,49.725,159.650
C03333=1020.390,306.023,-137.765,170.345,49.728,159.650
C03334=1020.383,305.775,-137.732,170.339,49.732,159.650
C03335=1020.376,305.528,-137.700,170.334,49.735,159.650
C03336=1020.369,305.280,-137.667,170.329,49.738,159.650
C03337=1020.363,305.032,-137.634,170.323,49.742,159.650
C03338=1020.355,304.784,-137.602,170.318,49.744,159.650
C03339=1020.349,304.536,-137.570,170.312,49.747,159.649
C03340=1020.342,304.289,-137.538,170.306,49.751,159.649
C03341=1020.336,304.041,-137.505,170.301,49.754,159.649
C03342=1020.329,303.794,-137.473,170.295,49.758,159.649
C03343=1020.322,303.545,-137.440,170.290,49.761,159.649
C03344=1020.316,303.297,-137.408,170.285,49.764,159.649
C03345=1020.309,303.050,-137.375,170.279,49.767,159.649
C03346=1020.303,302.802,-137.343,170.274,49.771,159.649
C03347=1020.296,302.555,-137.311,170.268,49.774,159.649
C03348=1020.290,302.307,-137.278,170.263,49.778,159.648
C03349=1020.284,302.059,-137.246,170.257,49.781,159.648
C03350=1020.277,301.812,-137.214,170.252,49.784,159.648
C03351=1020.270,301.563,-137.182,170.247,49.787,159.648
C03352=1020.263,301.315,-137.150,170.241,49.791,159.648
C03353=1020.257,301.068,-137.117,170.236,49.794,159.648
C03354=1020.251,300.820,-137.085,170.230,49.798,159.648
C03355=1020.244,300.572,-137.053,170.225,49.801,159.648
C03356=1020.238,300.324,-137.021,170.219,49.804,159.648
C03357=1020.231,300.077,-136.989,170.214,49.807,159.647
C03358=1020.225,299.829,-136.957,170.209,49.811,159.648
C03359=1020.218,299.581,-136.924,170.204,49.815,159.647
C03360=1020.212,299.333,-136.892,170.198,49.818,159.647
C03361=1020.206,299.086,-136.860,170.193,49.821,159.647
C03362=1020.199,298.838,-136.828,170.188,49.825,159.647
C03363=1020.193,298.589,-136.796,170.182,49.828,159.647
C03364=1020.186,298.342,-136.764,170.177,49.832,159.647
C03365=1020.180,298.094,-136.732,170.171,49.835,159.647
C03366=1020.174,297.846,-136.700,170.166,49.839,159.647
C03367=1020.167,297.598,-136.668,170.161,49.842,159.647
C03368=1020.161,297.350,-136.636,170.155,49.845,159.647
C03369=1020.154,297.102,-136.604,170.151,49.849,159.647
C03370=1020.148,296.855,-136.572,170.145,49.852,159.647
C03371=1020.141,296.607,-136.540,170.140,49.856,159.646
C03372=1020.136,296.359,-136.509,170.135,49.860,159.647
C03373=1020.129,296.112,-136.476,170.130,49.863,159.646
C03374=1020.123,295.864,-136.444,170.123,49.867,159.646
C03375=1020.117,295.616,-136.412,170.118,49.870,159.646
C03376=1020.110,295.368,-136.381,170.113,49.874,159.646
C03377=1020.104,295.119,-136.349,170.108,49.877,159.646
C03378=1020.097,294.872,-136.317,170.103,49.881,159.646
C03379=1020.092,294.625,-136.285,170.098,49.884,159.646
C03380=1020.086,294.376,-136.253,170.092,49.888,159.646
C03381=1020.079,294.129,-136.222,170.087,49.891,159.646
C03382=1020.073,293.880,-136.190,170.082,49.895,159.646
C03383=1020.067,293.649,-136.160,170.077,49.899,159.646
C03384=1020.061,293.418,-136.130,170.073,49.902,159.646
C03385=1020.055,293.186,-136.101,170.068,49.905,159.646
C03386=1020.049,292.955,-136.072,170.063,49.909,159.646
C03387=1020.043,292.724,-136.042,170.057,49.912,159.646
C03388=1020.037,292.492,-136.013,170.053,49.915,159.646
C03389=1020.031,292.260,-135.983,170.048,49.919,159.646
C03390=1020.025,292.029,-135.955,170.043,49.922,159.646
C03391=1020.019,291.781,-135.923,170.038,49.926,159.646
C03392=1020.013,291.533,-135.891,170.033,49.930,159.646
C03393=1020.006,291.285,-135.860,170.028,49.934,159.646
C03394=1019.999,291.037,-135.829,170.023,49.938,159.646
C03395=1019.993,290.790,-135.798,170.018,49.941,159.646
C03396=1019.987,290.542,-135.767,170.013,49.945,159.646
C03397=1019.980,290.294,-135.735,170.007,49.949,159.646
C03398=1019.974,290.045,-135.705,170.002,49.953,159.646
C03399=1019.968,289.798,-135.673,169.997,49.957,159.646
C03400=1019.961,289.550,-135.642,169.992,49.961,159.646
C03401=1019.955,289.301,-135.611,169.987,49.965,159.646
C03402=1019.948,289.053,-135.579,169.982,49.968,159.646
C03403=1019.942,288.806,-135.548,169.977,49.972,159.646
C03404=1019.936,288.558,-135.518,169.972,49.976,159.646
C03405=1019.929,288.310,-135.486,169.966,49.980,159.646
C03406=1019.923,288.062,-135.456,169.961,49.984,159.647
C03407=1019.916,287.814,-135.424,169.956,49.988,159.647
C03408=1019.910,287.566,-135.393,169.951,49.992,159.647
C03409=1019.904,287.318,-135.363,169.946,49.996,159.647
C03410=1019.897,287.070,-135.331,169.941,50.000,159.647
C03411=1019.891,286.823,-135.301,169.937,50.004,159.647
C03412=1019.885,286.574,-135.270,169.932,50.008,159.647
C03413=1019.878,286.326,-135.239,169.927,50.012,159.647
C03414=1019.872,286.078,-135.208,169.921,50.016,159.647
C03415=1019.866,285.830,-135.177,169.916,50.020,159.647
C03416=1019.859,285.582,-135.146,169.911,50.024,159.647
C03417=1019.853,285.335,-135.115,169.906,50.028,159.647
C03418=1019.847,285.086,-135.084,169.901,50.032,159.648
C03419=1019.841,284.838,-135.054,169.896,50.036,159.648
C03420=1019.834,284.590,-135.023,169.891,50.040,159.648
C03421=1019.828,284.343,-134.992,169.886,50.044,159.648
C03422=1019.822,284.094,-134.962,169.880,50.048,159.648
C03423=1019.815,283.847,-134.932,169.876,50.052,159.648
C03424=1019.809,283.598,-134.901,169.871,50.057,159.648
C03425=1019.802,283.350,-134.870,169.866,50.061,159.648
C03426=1019.796,283.102,-134.839,169.861,50.065,159.648
C03427=1019.789,282.854,-134.809,169.856,50.069,159.648
C03428=1019.783,282.606,-134.779,169.851,50.074,159.649
C03429=1019.777,282.358,-134.748,169.846,50.078,159.649
C03430=1019.771,282.110,-134.718,169.841,50.082,159.649
C03431=1019.765,281.861,-134.687,169.836,50.086,159.649
C03432=1019.758,281.614,-134.657,169.831,50.090,159.649
C03433=1019.752,281.366,-134.626,169.827,50.094,159.649
C03434=1019.746,281.118,-134.595,169.822,50.098,159.649
C03435=1019.739,280.870,-134.565,169.817,50.103,159.650
C03436=1019.733,280.622,-134.535,169.811,50.107,159.650
C03437=1019.727,280.374,-134.505,169.806,50.111,159.650
C03438=1019.721,280.126,-134.474,169.802,50.116,159.650
C03439=1019.715,279.878,-134.444,169.797,50.120,159.650
C03440=1019.708,279.629,-134.413,169.792,50.124,159.650
C03441=1019.702,279.382,-134.383,169.787,50.128,159.650
C03442=1019.696,279.134,-134.353,169.782,50.132,159.651
C03443=1019.690,278.909,-134.325,169.778,50.136,159.651
C03444=1019.685,278.683,-134.297,169.773,50.140,159.651
C03445=1019.679,278.458,-134.270,169.769,50.144,159.651
C03446=1019.673,278.232,-134.242,169.764,50.148,159.651
C03447=1019.668,278.007,-134.215,169.760,50.152,159.651
C03448=1019.662,277.781,-134.188,169.755,50.156,159.651
C03449=1019.657,277.556,-134.160,169.752,50.160,159.652
C03450=1019.651,277.330,-134.133,169.747,50.164,159.652
C03451=1019.645,277.083,-134.103,169.742,50.168,159.652
C03452=1019.638,276.834,-134.073,169.737,50.172,159.652
C03453=1019.632,276.587,-134.042,169.733,50.177,159.652
C03454=1019.627,276.339,-134.012,169.728,50.182,159.653
C03455=1019.620,276.090,-133.983,169.722,50.186,159.653
C03456=1019.614,275.842,-133.952,169.718,50.191,159.653
C03457=1019.607,275.595,-133.923,169.713,50.195,159.653
C03458=1019.601,275.346,-133.893,169.708,50.199,159.653
C03459=1019.595,275.098,-133.863,169.704,50.204,159.654
C03460=1019.589,274.850,-133.833,169.699,50.208,159.654
C03461=1019.582,274.601,-133.803,169.693,50.213,159.654
C03462=1019.576,274.354,-133.773,169.689,50.217,159.654
C03463=1019.570,274.105,-133.744,169.684,50.222,159.654
C03464=1019.564,273.858,-133.713,169.680,50.227,159.655
C03465=1019.557,273.609,-133.684,169.675,50.231,159.655
C03466=1019.552,273.361,-133.654,169.670,50.235,159.655
C03467=1019.545,273.113,-133.625,169.666,50.240,159.655
C03468=1019.539,272.865,-133.594,169.660,50.245,159.655
C03469=1019.533,272.616,-133.565,169.655,50.249,159.656
C03470=1019.527,272.368,-133.534,169.651,50.254,159.656
C03471=1019.521,272.120,-133.505,169.646,50.258,159.656
C03472=1019.515,271.872,-133.475,169.642,50.263,159.656
C03473=1019.508,271.624,-133.446,169.637,50.268,159.657
C03474=1019.502,271.375,-133.417,169.632,50.273,159.657
C03475=1019.496,271.128,-133.386,169.627,50.277,159.657
C03476=1019.490,270.879,-133.357,169.623,50.282,159.657
C03477=1019.484,270.632,-133.327,169.618,50.286,159.657
C03478=1019.477,270.383,-133.298,169.613,50.290,159.658
C03479=1019.472,270.135,-133.268,169.609,50.295,159.658
C03480=1019.465,269.886,-133.239,169.603,50.300,159.658
C03481=1019.459,269.639,-133.209,169.599,50.305,159.659
C03482=1019.453,269.390,-133.179,169.594,50.309,159.659
C03483=1019.447,269.142,-133.150,169.590,50.314,159.659
C03484=1019.440,268.895,-133.121,169.585,50.319,159.659
C03485=1019.435,268.646,-133.091,169.580,50.324,159.660
C03486=1019.428,268.398,-133.062,169.575,50.329,159.660
C03487=1019.422,268.150,-133.033,169.571,50.334,159.660
C03488=1019.416,267.902,-133.004,169.566,50.338,159.661
C03489=1019.410,267.653,-132.974,169.562,50.343,159.661
C03490=1019.404,267.404,-132.945,169.557,50.348,159.661
C03491=1019.397,267.157,-132.915,169.552,50.353,159.661
C03492=1019.391,266.909,-132.886,169.547,50.357,159.662
C03493=1019.385,266.660,-132.856,169.543,50.362,159.662
C03494=1019.379,266.412,-132.827,169.539,50.367,159.662
C03495=1019.373,266.164,-132.798,169.534,50.372,159.663
C03496=1019.367,265.916,-132.769,169.529,50.377,159.663
C03497=1019.360,265.668,-132.740,169.524,50.382,159.663
C03498=1019.355,265.419,-132.711,169.520,50.386,159.663
C03499=1019.349,265.171,-132.682,169.515,50.392,159.664
C03500=1019.342,264.923,-132.653,169.511,50.396,159.664
C03501=1019.336,264.675,-132.623,169.505,50.401,159.664
C03502=1019.330,264.427,-132.594,169.501,50.407,159.665
C03503=1019.324,264.203,-132.568,169.497,50.411,159.665
C03504=1019.319,263.980,-132.543,169.493,50.415,159.665
C03505=1019.314,263.757,-132.516,169.488,50.420,159.665
C03506=1019.308,263.535,-132.491,169.485,50.424,159.666
C03507=1019.302,263.311,-132.465,169.480,50.429,159.666
C03508=1019.297,263.088,-132.438,169.477,50.433,159.667
C03509=1019.292,262.865,-132.413,169.472,50.438,159.667
C03510=1019.286,262.642,-132.387,169.468,50.442,159.667
C03511=1019.280,262.394,-132.358,169.463,50.447,159.667
C03512=1019.274,262.146,-132.328,169.459,50.452,159.668
C03513=1019.267,261.897,-132.299,169.455,50.457,159.668
C03514=1019.261,261.649,-132.270,169.450,50.463,159.668
C03515=1019.255,261.400,-132.242,169.445,50.468,159.669
C03516=1019.249,261.153,-132.213,169.441,50.473,159.669
C03517=1019.243,260.905,-132.184,169.436,50.478,159.669
C03518=1019.237,260.656,-132.156,169.432,50.483,159.670
C03519=1019.232,260.408,-132.126,169.427,50.488,159.670
C03520=1019.226,260.160,-132.097,169.423,50.493,159.671
C03521=1019.220,259.911,-132.069,169.418,50.498,159.671
C03522=1019.213,259.663,-132.041,169.414,50.503,159.671
C03523=1019.207,259.414,-132.012,169.409,50.509,159.672
C03524=1019.200,259.166,-131.984,169.404,50.514,159.672
C03525=1019.194,258.918,-131.956,169.400,50.519,159.673
C03526=1019.188,258.670,-131.927,169.395,50.525,159.673
C03527=1019.181,258.422,-131.899,169.391,50.530,159.673
C03528=1019.175,258.174,-131.870,169.387,50.535,159.674
C03529=1019.169,257.925,-131.842,169.381,50.540,159.674
C03530=1019.163,257.677,-131.814,169.377,50.546,159.675
C03531=1019.156,257.428,-131.785,169.373,50.551,159.675
C03532=1019.150,257.180,-131.757,169.368,50.556,159.675
C03533=1019.144,256.932,-131.729,169.364,50.562,159.676
C03534=1019.138,256.684,-131.700,169.359,50.567,159.676
C03535=1019.132,256.435,-131.672,169.354,50.573,159.677
C03536=1019.125,256.187,-131.644,169.350,50.578,159.677
C03537=1019.119,255.938,-131.615,169.346,50.583,159.677
C03538=1019.113,255.690,-131.587,169.341,50.588,159.678
C03539=1019.107,255.442,-131.559,169.337,50.594,159.678
C03540=1019.101,255.194,-131.530,169.332,50.599,159.679
C03541=1019.095,254.945,-131.502,169.328,50.605,159.679
C03542=1019.088,254.697,-131.474,169.323,50.610,159.679
C03543=1019.083,254.449,-131.446,169.319,50.616,159.680
C03544=1019.077,254.200,-131.417,169.315,50.621,159.680
C03545=1019.070,253.952,-131.390,169.310,50.627,159.681
C03546=1019.064,253.703,-131.361,169.306,50.632,159.681
C03547=1019.059,253.455,-131.333,169.302,50.637,159.682
C03548=1019.052,253.207,-131.306,169.297,50.643,159.682
C03549=1019.046,252.958,-131.277,169.292,50.648,159.683
C03550=1019.040,252.710,-131.248,169.288,50.654,159.683
C03551=1019.034,252.462,-131.221,169.283,50.660,159.683
C03552=1019.028,252.213,-131.193,169.279,50.665,159.684
C03553=1019.022,251.965,-131.164,169.275,50.670,159.684
C03554=1019.016,251.717,-131.137,169.270,50.676,159.685
C03555=1019.010,251.468,-131.109,169.266,50.681,159.685
C03556=1019.003,251.220,-131.081,169.262,50.687,159.686
C03557=1018.998,250.972,-131.053,169.257,50.693,159.686
C03558=1018.992,250.723,-131.025,169.252,50.698,159.687
C03559=1018.985,250.474,-130.997,169.248,50.703,159.687
C03560=1018.980,250.226,-130.969,169.243,50.709,159.687
C03561=1018.974,249.978,-130.940,169.239,50.714,159.688
C03562=1018.967,249.729,-130.913,169.235,50.720,159.688
C03563=1018.962,249.506,-130.887,169.231,50.725,159.689
C03564=1018.957,249.282,-130.862,169.227,50.731,159.689
C03565=1018.951,249.058,-130.837,169.223,50.735,159.690
C03566=1018.946,248.834,-130.812,169.219,50.740,159.690
C03567=1018.941,248.610,-130.786,169.215,50.746,159.691
C03568=1018.935,248.386,-130.760,169.212,50.750,159.691
C03569=1018.930,248.163,-130.736,169.208,50.755,159.691
C03570=1018.925,247.939,-130.711,169.204,50.761,159.692
C03571=1018.919,247.690,-130.683,169.199,50.766,159.692
C03572=1018.913,247.442,-130.655,169.195,50.772,159.693
C03573=1018.907,247.193,-130.627,169.190,50.777,159.693
C03574=1018.901,246.946,-130.599,169.186,50.783,159.694
C03575=1018.895,246.696,-130.572,169.182,50.789,159.694
